Yaskawa INFORM job: A_ROOF_SIDE_0617_2_PAINT_29.JBI

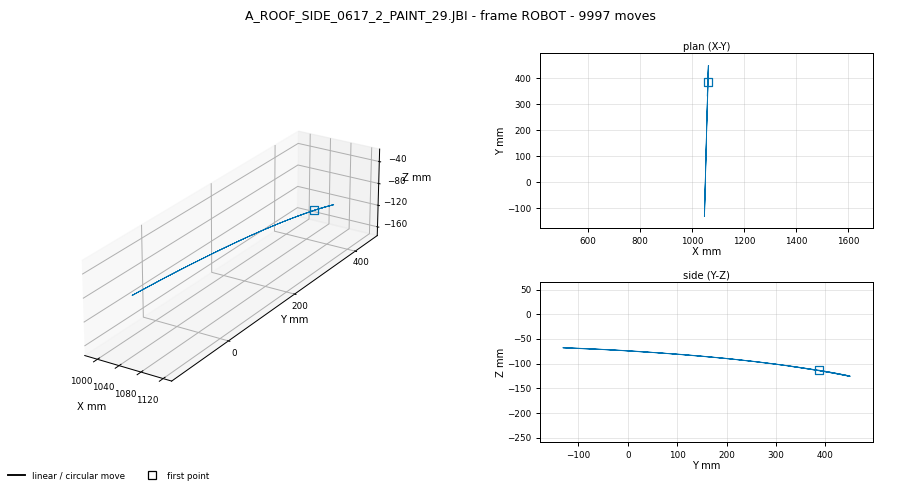
[picture p0: tool path of A_ROOF_SIDE_0617_2_PAINT_29.JBI in frame ROBOT, 9997 of 9997 moves have a stored position in this frame; points joined in program order, loops and branches not executed]
/JOB
//NAME A_ROOF_SIDE_0617_2_PAINT29
//POS
///NPOS 9997,0,0,0,0,0
///TOOL 1
///USER 0
///POSTYPE ROBOT
///RECTAN
///RCONF 1,0,0,0,0,0,0,0,0,0,0,0,0,0,0,0,0,0,0,0,0,0,0,0
C00000=1061.850,386.857,-113.195,174.714,36.908,156.968
C00001=1061.859,387.148,-113.243,174.721,36.916,156.970
C00002=1061.868,387.440,-113.291,174.727,36.924,156.972
C00003=1061.877,387.731,-113.339,174.733,36.933,156.974
C00004=1061.885,387.977,-113.380,174.739,36.940,156.976
C00005=1061.892,388.224,-113.421,174.745,36.947,156.978
C00006=1061.900,388.470,-113.462,174.750,36.954,156.979
C00007=1061.908,388.717,-113.503,174.756,36.961,156.981
C00008=1061.916,388.963,-113.543,174.761,36.968,156.983
C00009=1061.923,389.210,-113.585,174.766,36.975,156.985
C00010=1061.931,389.456,-113.625,174.773,36.983,156.986
C00011=1061.938,389.703,-113.667,174.778,36.990,156.988
C00012=1061.946,389.949,-113.707,174.783,36.997,156.990
C00013=1061.954,390.196,-113.748,174.789,37.004,156.992
C00014=1061.962,390.442,-113.789,174.794,37.012,156.994
C00015=1061.969,390.688,-113.830,174.801,37.019,156.995
C00016=1061.976,390.935,-113.872,174.806,37.026,156.997
C00017=1061.984,391.181,-113.913,174.812,37.034,156.999
C00018=1061.992,391.427,-113.954,174.817,37.041,157.001
C00019=1061.999,391.674,-113.995,174.822,37.048,157.003
C00020=1062.006,391.920,-114.037,174.829,37.056,157.005
C00021=1062.015,392.166,-114.078,174.834,37.063,157.006
C00022=1062.022,392.413,-114.119,174.840,37.071,157.008
C00023=1062.029,392.659,-114.160,174.845,37.078,157.010
C00024=1062.037,392.905,-114.202,174.852,37.086,157.012
C00025=1062.045,393.152,-114.243,174.857,37.093,157.014
C00026=1062.053,393.398,-114.285,174.863,37.100,157.016
C00027=1062.060,393.645,-114.326,174.868,37.108,157.017
C00028=1062.068,393.891,-114.368,174.875,37.116,157.019
C00029=1062.075,394.137,-114.410,174.880,37.123,157.021
C00030=1062.083,394.383,-114.452,174.886,37.131,157.023
C00031=1062.090,394.629,-114.494,174.892,37.139,157.025
C00032=1062.098,394.877,-114.535,174.898,37.146,157.027
C00033=1062.107,395.122,-114.576,174.903,37.154,157.029
C00034=1062.114,395.368,-114.618,174.910,37.161,157.031
C00035=1062.122,395.615,-114.660,174.916,37.170,157.033
C00036=1062.130,395.862,-114.702,174.921,37.177,157.035
C00037=1062.137,396.107,-114.744,174.928,37.185,157.037
C00038=1062.145,396.353,-114.786,174.933,37.192,157.039
C00039=1062.152,396.600,-114.827,174.939,37.200,157.041
C00040=1062.160,396.847,-114.869,174.945,37.208,157.042
C00041=1062.168,397.093,-114.911,174.951,37.216,157.044
C00042=1062.176,397.339,-114.954,174.957,37.223,157.046
C00043=1062.184,397.585,-114.996,174.963,37.232,157.048
C00044=1062.191,397.831,-115.038,174.969,37.240,157.050
C00045=1062.200,398.078,-115.080,174.974,37.247,157.052
C00046=1062.207,398.324,-115.122,174.981,37.255,157.054
C00047=1062.215,398.571,-115.164,174.987,37.263,157.056
C00048=1062.222,398.817,-115.207,174.993,37.271,157.058
C00049=1062.230,399.062,-115.249,174.999,37.279,157.060
C00050=1062.238,399.309,-115.292,175.005,37.287,157.062
C00051=1062.246,399.555,-115.334,175.011,37.295,157.064
C00052=1062.254,399.802,-115.376,175.017,37.303,157.066
C00053=1062.262,400.048,-115.418,175.024,37.311,157.068
C00054=1062.270,400.294,-115.461,175.029,37.319,157.070
C00055=1062.277,400.540,-115.503,175.036,37.327,157.073
C00056=1062.288,400.848,-115.556,175.043,37.337,157.075
C00057=1062.297,401.157,-115.609,175.051,37.348,157.078
C00058=1062.307,401.465,-115.663,175.059,37.358,157.080
C00059=1062.318,401.773,-115.716,175.067,37.368,157.083
C00060=1062.325,402.019,-115.760,175.073,37.376,157.085
C00061=1062.333,402.265,-115.802,175.079,37.385,157.087
C00062=1062.342,402.511,-115.845,175.086,37.393,157.089
C00063=1062.349,402.757,-115.887,175.092,37.401,157.091
C00064=1062.357,403.004,-115.930,175.099,37.410,157.094
C00065=1062.365,403.250,-115.973,175.104,37.418,157.096
C00066=1062.373,403.496,-116.015,175.111,37.426,157.098
C00067=1062.381,403.742,-116.059,175.117,37.435,157.100
C00068=1062.389,403.988,-116.102,175.124,37.443,157.102
C00069=1062.397,404.235,-116.146,175.130,37.451,157.104
C00070=1062.405,404.481,-116.188,175.136,37.460,157.106
C00071=1062.412,404.727,-116.231,175.143,37.468,157.109
C00072=1062.421,404.973,-116.274,175.149,37.477,157.111
C00073=1062.429,405.219,-116.317,175.156,37.485,157.113
C00074=1062.437,405.465,-116.361,175.162,37.494,157.115
C00075=1062.446,405.711,-116.404,175.169,37.503,157.117
C00076=1062.453,405.957,-116.447,175.176,37.511,157.120
C00077=1062.461,406.203,-116.491,175.182,37.520,157.122
C00078=1062.469,406.450,-116.534,175.188,37.529,157.124
C00079=1062.477,406.696,-116.577,175.194,37.537,157.126
C00080=1062.485,406.942,-116.620,175.201,37.546,157.129
C00081=1062.493,407.188,-116.665,175.208,37.555,157.131
C00082=1062.501,407.434,-116.708,175.215,37.564,157.133
C00083=1062.510,407.680,-116.751,175.221,37.572,157.135
C00084=1062.517,407.926,-116.795,175.228,37.581,157.138
C00085=1062.525,408.172,-116.839,175.235,37.590,157.140
C00086=1062.533,408.418,-116.882,175.241,37.599,157.142
C00087=1062.541,408.664,-116.926,175.248,37.608,157.145
C00088=1062.549,408.910,-116.970,175.255,37.616,157.147
C00089=1062.558,409.156,-117.013,175.261,37.625,157.149
C00090=1062.566,409.402,-117.058,175.268,37.634,157.151
C00091=1062.574,409.649,-117.101,175.275,37.643,157.154
C00092=1062.582,409.894,-117.146,175.282,37.652,157.156
C00093=1062.591,410.140,-117.189,175.288,37.661,157.158
C00094=1062.599,410.386,-117.233,175.295,37.670,157.161
C00095=1062.607,410.632,-117.277,175.302,37.679,157.163
C00096=1062.615,410.878,-117.320,175.310,37.688,157.165
C00097=1062.623,411.124,-117.365,175.317,37.697,157.168
C00098=1062.632,411.370,-117.409,175.323,37.706,157.170
C00099=1062.640,411.616,-117.454,175.330,37.716,157.173
C00100=1062.649,411.862,-117.497,175.337,37.725,157.175
C00101=1062.657,412.108,-117.541,175.344,37.734,157.177
C00102=1062.665,412.354,-117.586,175.351,37.743,157.180
C00103=1062.673,412.600,-117.630,175.358,37.752,157.182
C00104=1062.682,412.845,-117.674,175.365,37.762,157.185
C00105=1062.691,413.092,-117.719,175.372,37.771,157.187
C00106=1062.699,413.337,-117.763,175.379,37.780,157.190
C00107=1062.707,413.583,-117.807,175.386,37.790,157.192
C00108=1062.716,413.829,-117.851,175.394,37.799,157.194
C00109=1062.725,414.075,-117.896,175.401,37.808,157.197
C00110=1062.733,414.322,-117.941,175.408,37.818,157.199
C00111=1062.741,414.567,-117.985,175.415,37.827,157.202
C00112=1062.752,414.880,-118.042,175.424,37.839,157.205
C00113=1062.762,415.193,-118.099,175.434,37.852,157.208
C00114=1062.773,415.506,-118.156,175.443,37.864,157.212
C00115=1062.784,415.820,-118.214,175.452,37.876,157.215
C00116=1062.792,416.065,-118.258,175.460,37.886,157.217
C00117=1062.801,416.311,-118.303,175.467,37.896,157.220
C00118=1062.809,416.557,-118.348,175.474,37.905,157.223
C00119=1062.818,416.803,-118.393,175.482,37.915,157.225
C00120=1062.826,417.049,-118.438,175.489,37.925,157.228
C00121=1062.835,417.294,-118.483,175.497,37.935,157.230
C00122=1062.843,417.540,-118.528,175.504,37.945,157.233
C00123=1062.852,417.786,-118.573,175.511,37.954,157.236
C00124=1062.860,418.031,-118.618,175.519,37.964,157.238
C00125=1062.869,418.277,-118.664,175.526,37.974,157.241
C00126=1062.878,418.524,-118.709,175.534,37.984,157.243
C00127=1062.886,418.769,-118.754,175.541,37.994,157.246
C00128=1062.895,419.015,-118.799,175.549,38.004,157.249
C00129=1062.903,419.261,-118.845,175.557,38.014,157.251
C00130=1062.912,419.506,-118.890,175.565,38.024,157.254
C00131=1062.920,419.752,-118.935,175.572,38.034,157.257
C00132=1062.929,419.998,-118.981,175.580,38.043,157.259
C00133=1062.938,420.243,-119.026,175.587,38.054,157.262
C00134=1062.947,420.489,-119.072,175.595,38.064,157.265
C00135=1062.955,420.735,-119.117,175.604,38.074,157.268
C00136=1062.964,420.980,-119.163,175.611,38.084,157.270
C00137=1062.973,421.226,-119.210,175.619,38.095,157.273
C00138=1062.982,421.472,-119.255,175.626,38.105,157.276
C00139=1062.991,421.718,-119.300,175.635,38.116,157.279
C00140=1062.998,421.962,-119.347,175.643,38.125,157.282
C00141=1063.007,422.208,-119.392,175.650,38.136,157.284
C00142=1063.016,422.454,-119.438,175.658,38.146,157.287
C00143=1063.025,422.700,-119.484,175.666,38.157,157.290
C00144=1063.033,422.946,-119.530,175.674,38.167,157.293
C00145=1063.043,423.191,-119.576,175.682,38.178,157.296
C00146=1063.051,423.436,-119.623,175.691,38.188,157.299
C00147=1063.060,423.682,-119.669,175.698,38.199,157.301
C00148=1063.069,423.927,-119.715,175.706,38.210,157.304
C00149=1063.078,424.173,-119.761,175.715,38.220,157.307
C00150=1063.087,424.419,-119.807,175.723,38.230,157.310
C00151=1063.095,424.664,-119.854,175.731,38.241,157.313
C00152=1063.105,424.910,-119.900,175.739,38.252,157.316
C00153=1063.113,425.155,-119.946,175.747,38.263,157.319
C00154=1063.122,425.400,-119.993,175.756,38.274,157.322
C00155=1063.131,425.646,-120.039,175.764,38.284,157.325
C00156=1063.140,425.891,-120.085,175.773,38.295,157.328
C00157=1063.149,426.137,-120.133,175.780,38.306,157.331
C00158=1063.159,426.382,-120.179,175.789,38.317,157.334
C00159=1063.167,426.628,-120.225,175.797,38.328,157.337
C00160=1063.177,426.873,-120.272,175.806,38.339,157.340
C00161=1063.185,427.119,-120.318,175.814,38.350,157.343
C00162=1063.194,427.365,-120.365,175.823,38.361,157.346
C00163=1063.203,427.610,-120.413,175.831,38.372,157.349
C00164=1063.212,427.855,-120.459,175.840,38.383,157.352
C00165=1063.221,428.100,-120.506,175.849,38.394,157.355
C00166=1063.230,428.346,-120.554,175.857,38.405,157.358
C00167=1063.239,428.592,-120.600,175.866,38.417,157.361
C00168=1063.252,428.924,-120.664,175.877,38.432,157.365
C00169=1063.264,429.258,-120.728,175.889,38.447,157.370
C00170=1063.276,429.591,-120.792,175.902,38.463,157.374
C00171=1063.289,429.925,-120.856,175.913,38.478,157.378
C00172=1063.298,430.170,-120.904,175.922,38.489,157.381
C00173=1063.308,430.415,-120.951,175.931,38.501,157.384
C00174=1063.316,430.661,-120.998,175.940,38.512,157.388
C00175=1063.326,430.906,-121.046,175.948,38.524,157.391
C00176=1063.334,431.151,-121.093,175.958,38.536,157.394
C00177=1063.344,431.397,-121.141,175.967,38.547,157.397
C00178=1063.353,431.642,-121.189,175.976,38.559,157.401
C00179=1063.362,431.887,-121.237,175.984,38.570,157.404
C00180=1063.371,432.132,-121.284,175.993,38.582,157.407
C00181=1063.381,432.377,-121.332,176.003,38.594,157.411
C00182=1063.390,432.623,-121.380,176.012,38.606,157.414
C00183=1063.399,432.868,-121.428,176.021,38.618,157.417
C00184=1063.409,433.113,-121.476,176.031,38.629,157.420
C00185=1063.418,433.358,-121.524,176.040,38.641,157.424
C00186=1063.427,433.603,-121.572,176.049,38.653,157.427
C00187=1063.437,433.849,-121.619,176.059,38.665,157.431
C00188=1063.446,434.094,-121.668,176.068,38.677,157.434
C00189=1063.455,434.339,-121.715,176.077,38.689,157.437
C00190=1063.465,434.584,-121.764,176.087,38.701,157.441
C00191=1063.475,434.829,-121.812,176.096,38.714,157.444
C00192=1063.484,435.074,-121.860,176.106,38.726,157.448
C00193=1063.493,435.318,-121.908,176.115,38.738,157.451
C00194=1063.502,435.564,-121.957,176.124,38.750,157.454
C00195=1063.512,435.809,-122.005,176.134,38.763,157.458
C00196=1063.522,436.054,-122.054,176.144,38.775,157.462
C00197=1063.531,436.299,-122.102,176.153,38.787,157.465
C00198=1063.541,436.544,-122.151,176.163,38.799,157.469
C00199=1063.551,436.789,-122.199,176.173,38.812,157.472
C00200=1063.561,437.034,-122.248,176.183,38.824,157.476
C00201=1063.570,437.279,-122.296,176.192,38.837,157.479
C00202=1063.579,437.524,-122.346,176.202,38.849,157.483
C00203=1063.589,437.769,-122.394,176.212,38.862,157.486
C00204=1063.599,438.014,-122.443,176.222,38.874,157.490
C00205=1063.609,438.259,-122.492,176.232,38.887,157.494
C00206=1063.618,438.504,-122.541,176.242,38.900,157.497
C00207=1063.628,438.749,-122.589,176.251,38.912,157.501
C00208=1063.639,438.994,-122.639,176.262,38.925,157.505
C00209=1063.648,439.239,-122.688,176.272,38.938,157.508
C00210=1063.658,439.484,-122.737,176.282,38.951,157.512
C00211=1063.667,439.729,-122.786,176.292,38.964,157.516
C00212=1063.677,439.973,-122.836,176.302,38.977,157.520
C00213=1063.687,440.218,-122.885,176.313,38.990,157.523
C00214=1063.696,440.464,-122.935,176.323,39.003,157.527
C00215=1063.706,440.708,-122.984,176.334,39.016,157.531
C00216=1063.717,440.952,-123.033,176.344,39.029,157.535
C00217=1063.726,441.198,-123.083,176.354,39.042,157.538
C00218=1063.737,441.442,-123.132,176.364,39.056,157.542
C00219=1063.746,441.687,-123.182,176.375,39.069,157.546
C00220=1063.756,441.932,-123.232,176.385,39.082,157.550
C00221=1063.766,442.176,-123.282,176.396,39.095,157.554
C00222=1063.776,442.421,-123.331,176.407,39.109,157.558
C00223=1063.786,442.666,-123.381,176.417,39.122,157.562
C00224=1063.800,442.997,-123.449,176.432,39.141,157.567
C00225=1063.813,443.330,-123.517,176.446,39.159,157.573
C00226=1063.827,443.662,-123.585,176.461,39.177,157.578
C00227=1063.841,443.993,-123.652,176.477,39.196,157.583
C00228=1063.851,444.238,-123.703,176.487,39.209,157.587
C00229=1063.860,444.483,-123.753,176.498,39.223,157.592
C00230=1063.871,444.727,-123.804,176.509,39.237,157.596
C00231=1063.881,444.972,-123.854,176.520,39.251,157.600
C00232=1063.891,445.217,-123.904,176.532,39.265,157.604
C00233=1063.902,445.461,-123.955,176.543,39.279,157.608
C00234=1063.912,445.706,-124.006,176.554,39.293,157.612
C00235=1063.922,445.950,-124.056,176.566,39.307,157.616
C00236=1063.932,446.194,-124.106,176.576,39.321,157.620
C00237=1063.943,446.439,-124.157,176.588,39.335,157.625
C00238=1063.953,446.684,-124.208,176.600,39.349,157.629
C00239=1063.963,446.929,-124.259,176.611,39.364,157.633
C00240=1063.974,447.172,-124.310,176.622,39.378,157.637
C00241=1063.984,447.415,-124.360,176.634,39.392,157.642
C00242=1063.995,447.660,-124.411,176.645,39.406,157.646
C00243=1064.006,447.904,-124.461,176.657,39.420,157.650
C00244=1064.019,448.147,-124.510,176.669,39.434,157.654
C00245=1064.032,448.391,-124.559,176.681,39.447,157.658
C00246=1064.046,448.636,-124.607,176.693,39.460,157.662
C00247=1064.062,448.881,-124.655,176.704,39.473,157.666
C00248=1064.078,449.126,-124.702,176.716,39.486,157.670
C00249=1064.096,449.371,-124.748,176.729,39.498,157.674
C00250=1064.114,449.616,-124.793,176.740,39.510,157.677
C00251=1064.133,449.862,-124.838,176.752,39.522,157.681
C00252=1063.796,449.868,-125.107,176.744,39.644,157.714
C00253=1063.776,449.622,-125.063,176.733,39.632,157.711
C00254=1063.758,449.378,-125.017,176.720,39.621,157.707
C00255=1063.740,449.132,-124.971,176.708,39.608,157.703
C00256=1063.724,448.888,-124.924,176.696,39.596,157.699
C00257=1063.709,448.643,-124.877,176.684,39.583,157.695
C00258=1063.693,448.398,-124.828,176.672,39.570,157.691
C00259=1063.680,448.154,-124.780,176.660,39.557,157.687
C00260=1063.668,447.911,-124.731,176.648,39.543,157.683
C00261=1063.657,447.694,-124.686,176.637,39.531,157.679
C00262=1063.648,447.478,-124.642,176.627,39.518,157.676
C00263=1063.638,447.262,-124.596,176.617,39.506,157.672
C00264=1063.629,447.047,-124.551,176.606,39.493,157.668
C00265=1063.620,446.830,-124.507,176.596,39.480,157.664
C00266=1063.611,446.615,-124.462,176.586,39.468,157.661
C00267=1063.601,446.399,-124.417,176.576,39.455,157.657
C00268=1063.592,446.184,-124.372,176.566,39.443,157.653
C00269=1063.582,445.939,-124.321,176.555,39.429,157.649
C00270=1063.571,445.695,-124.271,176.543,39.415,157.645
C00271=1063.561,445.450,-124.220,176.532,39.401,157.641
C00272=1063.552,445.205,-124.170,176.521,39.387,157.637
C00273=1063.541,444.961,-124.120,176.510,39.373,157.632
C00274=1063.530,444.716,-124.069,176.498,39.360,157.628
C00275=1063.521,444.472,-124.018,176.487,39.346,157.624
C00276=1063.510,444.227,-123.969,176.476,39.332,157.620
C00277=1063.495,443.858,-123.892,176.459,39.311,157.614
C00278=1063.480,443.489,-123.817,176.442,39.291,157.608
C00279=1063.464,443.120,-123.741,176.427,39.271,157.602
C00280=1063.449,442.750,-123.665,176.410,39.250,157.596
C00281=1063.439,442.505,-123.616,176.399,39.237,157.592
C00282=1063.429,442.260,-123.566,176.389,39.224,157.588
C00283=1063.419,442.016,-123.516,176.378,39.210,157.584
C00284=1063.409,441.771,-123.465,176.367,39.197,157.580
C00285=1063.399,441.527,-123.416,176.357,39.184,157.576
C00286=1063.390,441.282,-123.366,176.346,39.170,157.573
C00287=1063.379,441.037,-123.317,176.335,39.157,157.569
C00288=1063.370,440.792,-123.267,176.325,39.144,157.565
C00289=1063.360,440.547,-123.218,176.314,39.131,157.561
C00290=1063.349,440.302,-123.169,176.304,39.118,157.557
C00291=1063.340,440.058,-123.119,176.294,39.105,157.554
C00292=1063.330,439.813,-123.070,176.284,39.092,157.550
C00293=1063.320,439.567,-123.020,176.273,39.080,157.546
C00294=1063.310,439.323,-122.971,176.263,39.066,157.542
C00295=1063.300,439.078,-122.922,176.252,39.054,157.539
C00296=1063.291,438.833,-122.873,176.243,39.041,157.535
C00297=1063.281,438.588,-122.824,176.233,39.028,157.531
C00298=1063.271,438.344,-122.775,176.222,39.015,157.527
C00299=1063.262,438.099,-122.726,176.212,39.003,157.524
C00300=1063.252,437.854,-122.676,176.203,38.990,157.520
C00301=1063.242,437.609,-122.628,176.192,38.978,157.517
C00302=1063.232,437.364,-122.579,176.182,38.965,157.513
C00303=1063.222,437.119,-122.530,176.173,38.952,157.509
C00304=1063.212,436.874,-122.482,176.162,38.940,157.506
C00305=1063.203,436.628,-122.433,176.153,38.928,157.502
C00306=1063.194,436.383,-122.384,176.143,38.915,157.499
C00307=1063.184,436.138,-122.336,176.134,38.903,157.495
C00308=1063.174,435.894,-122.287,176.124,38.891,157.492
C00309=1063.164,435.649,-122.239,176.114,38.879,157.488
C00310=1063.155,435.404,-122.190,176.104,38.867,157.485
C00311=1063.145,435.158,-122.142,176.094,38.854,157.481
C00312=1063.136,434.914,-122.094,176.085,38.842,157.478
C00313=1063.126,434.669,-122.046,176.076,38.830,157.474
C00314=1063.117,434.423,-121.998,176.066,38.818,157.471
C00315=1063.107,434.178,-121.949,176.057,38.806,157.468
C00316=1063.098,433.933,-121.900,176.047,38.794,157.464
C00317=1063.089,433.688,-121.853,176.038,38.782,157.461
C00318=1063.079,433.443,-121.804,176.029,38.770,157.457
C00319=1063.070,433.197,-121.756,176.019,38.759,157.454
C00320=1063.061,432.953,-121.709,176.010,38.746,157.451
C00321=1063.051,432.708,-121.661,176.001,38.735,157.447
C00322=1063.042,432.462,-121.613,175.991,38.723,157.444
C00323=1063.033,432.217,-121.565,175.982,38.711,157.441
C00324=1063.024,431.971,-121.517,175.973,38.699,157.437
C00325=1063.014,431.727,-121.469,175.964,38.688,157.434
C00326=1063.005,431.482,-121.421,175.954,38.676,157.431
C00327=1062.996,431.236,-121.374,175.945,38.664,157.428
C00328=1062.987,430.991,-121.326,175.937,38.653,157.424
C00329=1062.977,430.746,-121.278,175.928,38.641,157.421
C00330=1062.968,430.501,-121.231,175.919,38.630,157.418
C00331=1062.959,430.255,-121.184,175.909,38.619,157.415
C00332=1062.950,430.010,-121.137,175.900,38.607,157.411
C00333=1062.937,429.675,-121.072,175.889,38.592,157.407
C00334=1062.924,429.339,-121.008,175.877,38.576,157.403
C00335=1062.912,429.004,-120.943,175.864,38.561,157.399
C00336=1062.899,428.668,-120.878,175.852,38.545,157.394
C00337=1062.890,428.423,-120.832,175.844,38.534,157.391
C00338=1062.882,428.178,-120.784,175.835,38.523,157.388
C00339=1062.872,427.932,-120.738,175.826,38.512,157.385
C00340=1062.863,427.687,-120.690,175.818,38.501,157.382
C00341=1062.854,427.442,-120.643,175.809,38.490,157.379
C00342=1062.846,427.196,-120.597,175.801,38.479,157.376
C00343=1062.836,426.951,-120.549,175.792,38.468,157.373
C00344=1062.827,426.705,-120.503,175.784,38.457,157.370
C00345=1062.818,426.460,-120.457,175.775,38.446,157.367
C00346=1062.809,426.215,-120.410,175.766,38.435,157.364
C00347=1062.801,425.969,-120.363,175.759,38.424,157.361
C00348=1062.791,425.723,-120.317,175.750,38.414,157.358
C00349=1062.782,425.478,-120.270,175.742,38.403,157.355
C00350=1062.773,425.233,-120.224,175.733,38.392,157.352
C00351=1062.764,424.987,-120.178,175.725,38.382,157.349
C00352=1062.755,424.742,-120.131,175.716,38.371,157.346
C00353=1062.746,424.497,-120.085,175.708,38.360,157.343
C00354=1062.737,424.251,-120.038,175.700,38.349,157.340
C00355=1062.728,424.005,-119.993,175.692,38.339,157.337
C00356=1062.720,423.760,-119.946,175.684,38.328,157.334
C00357=1062.710,423.515,-119.900,175.675,38.318,157.332
C00358=1062.702,423.268,-119.854,175.668,38.307,157.329
C00359=1062.693,423.023,-119.808,175.660,38.297,157.326
C00360=1062.684,422.778,-119.761,175.651,38.286,157.323
C00361=1062.675,422.532,-119.715,175.644,38.276,157.320
C00362=1062.666,422.287,-119.669,175.635,38.265,157.317
C00363=1062.658,422.041,-119.623,175.627,38.255,157.315
C00364=1062.649,421.795,-119.577,175.620,38.245,157.312
C00365=1062.640,421.549,-119.531,175.611,38.235,157.309
C00366=1062.631,421.303,-119.486,175.603,38.224,157.306
C00367=1062.623,421.059,-119.439,175.596,38.214,157.303
C00368=1062.614,420.813,-119.394,175.588,38.204,157.301
C00369=1062.605,420.567,-119.349,175.580,38.193,157.298
C00370=1062.597,420.321,-119.303,175.572,38.183,157.295
C00371=1062.588,420.075,-119.257,175.564,38.174,157.292
C00372=1062.579,419.829,-119.212,175.557,38.163,157.290
C00373=1062.571,419.584,-119.167,175.548,38.153,157.287
C00374=1062.562,419.338,-119.121,175.541,38.143,157.284
C00375=1062.554,419.092,-119.075,175.533,38.133,157.282
C00376=1062.545,418.846,-119.030,175.526,38.123,157.279
C00377=1062.536,418.601,-118.985,175.518,38.113,157.276
C00378=1062.527,418.355,-118.939,175.511,38.103,157.273
C00379=1062.518,418.110,-118.894,175.502,38.094,157.271
C00380=1062.510,417.864,-118.849,175.495,38.084,157.268
C00381=1062.501,417.618,-118.804,175.487,38.074,157.266
C00382=1062.493,417.373,-118.759,175.480,38.064,157.263
C00383=1062.485,417.127,-118.713,175.473,38.055,157.260
C00384=1062.476,416.880,-118.668,175.465,38.045,157.258
C00385=1062.468,416.635,-118.623,175.458,38.035,157.255
C00386=1062.459,416.389,-118.578,175.450,38.025,157.253
C00387=1062.451,416.144,-118.534,175.443,38.016,157.250
C00388=1062.442,415.898,-118.488,175.436,38.006,157.247
C00389=1062.432,415.583,-118.431,175.426,37.994,157.244
C00390=1062.420,415.268,-118.374,175.416,37.981,157.241
C00391=1062.410,414.953,-118.316,175.407,37.969,157.238
C00392=1062.399,414.638,-118.259,175.398,37.957,157.234
C00393=1062.391,414.392,-118.214,175.390,37.948,157.232
C00394=1062.383,414.146,-118.169,175.383,37.938,157.229
C00395=1062.373,413.900,-118.125,175.376,37.929,157.227
C00396=1062.365,413.654,-118.081,175.369,37.920,157.225
C00397=1062.356,413.408,-118.036,175.362,37.910,157.222
C00398=1062.348,413.162,-117.992,175.355,37.901,157.220
C00399=1062.340,412.916,-117.948,175.348,37.892,157.217
C00400=1062.331,412.670,-117.904,175.341,37.882,157.215
C00401=1062.323,412.424,-117.859,175.333,37.873,157.212
C00402=1062.315,412.179,-117.815,175.326,37.864,157.210
C00403=1062.306,411.932,-117.770,175.319,37.855,157.207
C00404=1062.297,411.687,-117.726,175.312,37.846,157.205
C00405=1062.289,411.441,-117.682,175.305,37.836,157.203
C00406=1062.281,411.195,-117.638,175.298,37.827,157.200
C00407=1062.273,410.949,-117.594,175.292,37.818,157.198
C00408=1062.264,410.703,-117.550,175.284,37.809,157.195
C00409=1062.256,410.457,-117.506,175.277,37.800,157.193
C00410=1062.248,410.211,-117.462,175.270,37.791,157.191
C00411=1062.239,409.965,-117.418,175.263,37.782,157.188
C00412=1062.231,409.719,-117.374,175.257,37.773,157.186
C00413=1062.223,409.473,-117.330,175.250,37.764,157.184
C00414=1062.215,409.227,-117.286,175.243,37.755,157.181
C00415=1062.206,408.981,-117.243,175.236,37.746,157.179
C00416=1062.198,408.735,-117.198,175.229,37.738,157.177
C00417=1062.190,408.488,-117.155,175.223,37.729,157.174
C00418=1062.182,408.243,-117.111,175.216,37.720,157.172
C00419=1062.174,407.997,-117.067,175.209,37.711,157.170
C00420=1062.166,407.750,-117.024,175.202,37.702,157.168
C00421=1062.157,407.505,-116.980,175.196,37.694,157.165
C00422=1062.150,407.259,-116.936,175.189,37.685,157.163
C00423=1062.142,407.013,-116.893,175.182,37.676,157.161
C00424=1062.134,406.767,-116.850,175.176,37.668,157.159
C00425=1062.126,406.520,-116.806,175.169,37.659,157.156
C00426=1062.117,406.275,-116.763,175.162,37.650,157.154
C00427=1062.110,406.029,-116.719,175.156,37.642,157.152
C00428=1062.102,405.782,-116.675,175.150,37.633,157.150
C00429=1062.093,405.536,-116.632,175.143,37.624,157.147
C00430=1062.086,405.290,-116.589,175.137,37.616,157.145
C00431=1062.078,405.045,-116.546,175.130,37.607,157.143
C00432=1062.069,404.798,-116.503,175.123,37.599,157.141
C00433=1062.061,404.552,-116.459,175.117,37.591,157.139
C00434=1062.053,404.306,-116.416,175.110,37.582,157.136
C00435=1062.045,404.059,-116.374,175.104,37.574,157.134
C00436=1062.038,403.814,-116.331,175.098,37.565,157.132
C00437=1062.030,403.567,-116.287,175.091,37.557,157.130
C00438=1062.021,403.321,-116.244,175.085,37.548,157.128
C00439=1062.013,403.075,-116.202,175.078,37.540,157.126
C00440=1062.006,402.829,-116.159,175.072,37.532,157.123
C00441=1061.997,402.583,-116.116,175.066,37.523,157.121
C00442=1061.989,402.336,-116.073,175.059,37.515,157.119
C00443=1061.982,402.091,-116.030,175.053,37.507,157.117
C00444=1061.974,401.844,-115.988,175.046,37.499,157.115
C00445=1061.964,401.534,-115.934,175.038,37.489,157.112
C00446=1061.954,401.224,-115.880,175.031,37.478,157.110
C00447=1061.944,400.914,-115.827,175.023,37.468,157.107
C00448=1061.933,400.604,-115.773,175.016,37.458,157.105
C00449=1061.925,400.358,-115.730,175.009,37.450,157.102
C00450=1061.918,400.112,-115.688,175.003,37.441,157.100
C00451=1061.910,399.865,-115.646,174.996,37.433,157.098
C00452=1061.902,399.620,-115.603,174.991,37.425,157.096
C00453=1061.894,399.373,-115.561,174.984,37.418,157.094
C00454=1061.886,399.127,-115.519,174.978,37.410,157.092
C00455=1061.878,398.881,-115.476,174.972,37.402,157.090
C00456=1061.870,398.635,-115.434,174.966,37.394,157.088
C00457=1061.863,398.388,-115.391,174.959,37.386,157.086
C00458=1061.855,398.142,-115.349,174.954,37.378,157.084
C00459=1061.847,397.896,-115.306,174.948,37.370,157.082
C00460=1061.839,397.650,-115.265,174.942,37.362,157.080
C00461=1061.832,397.404,-115.223,174.936,37.354,157.078
C00462=1061.823,397.157,-115.180,174.929,37.346,157.076
C00463=1061.816,396.911,-115.138,174.924,37.339,157.074
C00464=1061.808,396.664,-115.096,174.918,37.331,157.072
C00465=1061.800,396.418,-115.055,174.912,37.323,157.070
C00466=1061.793,396.172,-115.013,174.906,37.315,157.068
C00467=1061.785,395.925,-114.971,174.899,37.308,157.066
C00468=1061.777,395.679,-114.929,174.894,37.300,157.065
C00469=1061.769,395.433,-114.887,174.888,37.293,157.063
C00470=1061.762,395.187,-114.845,174.882,37.284,157.061
C00471=1061.753,394.940,-114.804,174.876,37.277,157.059
C00472=1061.746,394.694,-114.762,174.871,37.269,157.057
C00473=1061.738,394.448,-114.721,174.864,37.262,157.055
C00474=1061.731,394.202,-114.679,174.859,37.254,157.053
C00475=1061.723,393.955,-114.636,174.853,37.247,157.051
C00476=1061.715,393.708,-114.595,174.847,37.239,157.049
C00477=1061.708,393.462,-114.553,174.841,37.232,157.047
C00478=1061.700,393.216,-114.512,174.836,37.224,157.046
C00479=1061.692,392.970,-114.471,174.829,37.216,157.044
C00480=1061.685,392.724,-114.429,174.824,37.209,157.042
C00481=1061.677,392.477,-114.387,174.818,37.202,157.040
C00482=1061.669,392.230,-114.346,174.813,37.194,157.038
C00483=1061.661,391.984,-114.305,174.806,37.187,157.036
C00484=1061.654,391.738,-114.263,174.801,37.179,157.034
C00485=1061.646,391.492,-114.222,174.795,37.172,157.033
C00486=1061.639,391.245,-114.181,174.789,37.164,157.031
C00487=1061.631,390.999,-114.139,174.783,37.157,157.029
C00488=1061.623,390.753,-114.098,174.778,37.150,157.027
C00489=1061.616,390.506,-114.057,174.773,37.143,157.025
C00490=1061.608,390.260,-114.016,174.766,37.135,157.023
C00491=1061.601,390.013,-113.975,174.761,37.128,157.022
C00492=1061.593,389.767,-113.934,174.755,37.121,157.020
C00493=1061.586,389.520,-113.893,174.750,37.114,157.018
C00494=1061.578,389.274,-113.853,174.745,37.106,157.016
C00495=1061.570,389.027,-113.811,174.738,37.099,157.014
C00496=1061.562,388.781,-113.771,174.733,37.092,157.013
C00497=1061.555,388.535,-113.729,174.727,37.085,157.011
C00498=1061.547,388.288,-113.689,174.722,37.078,157.009
C00499=1061.540,388.042,-113.648,174.717,37.071,157.007
C00500=1061.532,387.795,-113.607,174.710,37.064,157.006
C00501=1061.523,387.502,-113.558,174.704,37.055,157.004
C00502=1061.514,387.210,-113.511,174.698,37.047,157.001
C00503=1061.505,386.917,-113.461,174.691,37.039,156.999
C00504=1061.496,386.623,-113.413,174.685,37.030,156.997
C00505=1061.488,386.377,-113.373,174.679,37.023,156.996
C00506=1061.480,386.130,-113.331,174.674,37.016,156.994
C00507=1061.473,385.884,-113.292,174.668,37.009,156.992
C00508=1061.465,385.638,-113.251,174.663,37.002,156.990
C00509=1061.458,385.390,-113.211,174.657,36.996,156.989
C00510=1061.450,385.144,-113.170,174.652,36.988,156.987
C00511=1061.444,384.898,-113.129,174.647,36.981,156.985
C00512=1061.436,384.651,-113.089,174.641,36.975,156.984
C00513=1061.428,384.405,-113.049,174.636,36.968,156.982
C00514=1061.421,384.158,-113.008,174.631,36.961,156.980
C00515=1061.413,383.912,-112.968,174.626,36.954,156.979
C00516=1061.406,383.665,-112.927,174.619,36.947,156.977
C00517=1061.399,383.418,-112.887,174.614,36.940,156.975
C00518=1061.391,383.173,-112.847,174.609,36.933,156.974
C00519=1061.384,382.925,-112.807,174.604,36.927,156.972
C00520=1061.377,382.678,-112.767,174.599,36.920,156.970
C00521=1061.369,382.433,-112.726,174.593,36.913,156.969
C00522=1061.362,382.186,-112.686,174.588,36.906,156.967
C00523=1061.355,381.939,-112.646,174.583,36.899,156.965
C00524=1061.347,381.693,-112.606,174.578,36.893,156.964
C00525=1061.340,381.446,-112.565,174.573,36.886,156.962
C00526=1061.333,381.200,-112.526,174.568,36.879,156.960
C00527=1061.325,380.953,-112.486,174.562,36.873,156.959
C00528=1061.318,380.706,-112.445,174.557,36.866,156.957
C00529=1061.311,380.459,-112.406,174.552,36.859,156.956
C00530=1061.303,380.212,-112.366,174.546,36.853,156.954
C00531=1061.296,379.966,-112.326,174.541,36.846,156.952
C00532=1061.289,379.719,-112.286,174.536,36.840,156.951
C00533=1061.281,379.472,-112.246,174.530,36.833,156.949
C00534=1061.274,379.226,-112.207,174.525,36.826,156.948
C00535=1061.266,378.979,-112.167,174.520,36.820,156.946
C00536=1061.259,378.733,-112.127,174.515,36.813,156.945
C00537=1061.251,378.486,-112.087,174.510,36.807,156.943
C00538=1061.244,378.239,-112.048,174.505,36.801,156.941
C00539=1061.237,377.993,-112.009,174.500,36.794,156.940
C00540=1061.230,377.746,-111.969,174.495,36.787,156.938
C00541=1061.222,377.499,-111.929,174.490,36.781,156.937
C00542=1061.215,377.253,-111.890,174.484,36.775,156.935
C00543=1061.207,377.006,-111.850,174.479,36.768,156.934
C00544=1061.200,376.759,-111.811,174.475,36.762,156.932
C00545=1061.193,376.513,-111.771,174.470,36.756,156.931
C00546=1061.186,376.266,-111.732,174.465,36.749,156.929
C00547=1061.179,376.020,-111.692,174.460,36.743,156.928
C00548=1061.171,375.772,-111.653,174.455,36.736,156.926
C00549=1061.164,375.526,-111.614,174.450,36.730,156.925
C00550=1061.157,375.279,-111.575,174.445,36.724,156.923
C00551=1061.149,375.032,-111.535,174.440,36.718,156.921
C00552=1061.143,374.785,-111.496,174.435,36.711,156.920
C00553=1061.136,374.539,-111.457,174.430,36.705,156.918
C00554=1061.128,374.292,-111.417,174.425,36.698,156.917
C00555=1061.121,374.045,-111.378,174.420,36.692,156.915
C00556=1061.114,373.799,-111.339,174.415,36.686,156.914
C00557=1061.107,373.537,-111.297,174.410,36.680,156.912
C00558=1061.099,373.274,-111.256,174.404,36.673,156.911
C00559=1061.092,373.012,-111.214,174.399,36.666,156.909
C00560=1061.084,372.751,-111.173,174.394,36.660,156.908
C00561=1061.076,372.503,-111.134,174.389,36.653,156.906
C00562=1061.069,372.257,-111.095,174.384,36.647,156.905
C00563=1061.062,372.010,-111.056,174.379,36.641,156.903
C00564=1061.056,371.763,-111.017,174.375,36.635,156.902
C00565=1061.048,371.516,-110.978,174.370,36.629,156.900
C00566=1061.041,371.269,-110.940,174.365,36.623,156.899
C00567=1061.033,371.023,-110.901,174.360,36.617,156.897
C00568=1061.026,370.776,-110.862,174.355,36.610,156.896
C00569=1061.019,370.529,-110.823,174.350,36.604,156.894
C00570=1061.011,370.282,-110.784,174.345,36.598,156.893
C00571=1061.004,370.035,-110.745,174.341,36.593,156.892
C00572=1060.997,369.788,-110.707,174.337,36.587,156.890
C00573=1060.990,369.541,-110.669,174.332,36.580,156.889
C00574=1060.983,369.294,-110.630,174.327,36.574,156.887
C00575=1060.976,369.047,-110.591,174.322,36.568,156.886
C00576=1060.968,368.800,-110.553,174.317,36.562,156.884
C00577=1060.962,368.554,-110.514,174.312,36.557,156.883
C00578=1060.954,368.307,-110.476,174.307,36.551,156.882
C00579=1060.947,368.060,-110.437,174.303,36.544,156.880
C00580=1060.941,367.813,-110.399,174.298,36.539,156.879
C00581=1060.933,367.566,-110.361,174.294,36.533,156.878
C00582=1060.926,367.319,-110.322,174.289,36.527,156.876
C00583=1060.919,367.073,-110.283,174.284,36.521,156.875
C00584=1060.912,366.826,-110.245,174.279,36.515,156.873
C00585=1060.906,366.579,-110.207,174.275,36.509,156.872
C00586=1060.898,366.332,-110.168,174.270,36.503,156.871
C00587=1060.891,366.085,-110.130,174.265,36.497,156.869
C00588=1060.884,365.838,-110.092,174.261,36.492,156.868
C00589=1060.877,365.591,-110.054,174.256,36.486,156.866
C00590=1060.870,365.344,-110.016,174.252,36.480,156.865
C00591=1060.863,365.097,-109.977,174.247,36.474,156.864
C00592=1060.856,364.850,-109.939,174.242,36.468,156.862
C00593=1060.849,364.603,-109.901,174.238,36.462,156.861
C00594=1060.842,364.356,-109.862,174.233,36.457,156.860
C00595=1060.835,364.109,-109.825,174.229,36.451,156.858
C00596=1060.828,363.862,-109.786,174.224,36.445,156.857
C00597=1060.821,363.615,-109.748,174.219,36.439,156.856
C00598=1060.814,363.368,-109.711,174.215,36.434,156.854
C00599=1060.807,363.121,-109.672,174.210,36.428,156.853
C00600=1060.800,362.875,-109.635,174.206,36.422,156.852
C00601=1060.793,362.627,-109.597,174.201,36.416,156.850
C00602=1060.786,362.380,-109.560,174.197,36.411,156.849
C00603=1060.779,362.133,-109.521,174.192,36.405,156.848
C00604=1060.772,361.886,-109.483,174.188,36.400,156.846
C00605=1060.765,361.639,-109.446,174.183,36.394,156.845
C00606=1060.758,361.392,-109.408,174.178,36.389,156.844
C00607=1060.751,361.145,-109.370,174.174,36.383,156.842
C00608=1060.744,360.898,-109.333,174.170,36.377,156.841
C00609=1060.737,360.652,-109.295,174.165,36.372,156.840
C00610=1060.730,360.407,-109.258,174.161,36.366,156.839
C00611=1060.723,360.162,-109.220,174.156,36.361,156.837
C00612=1060.716,359.916,-109.183,174.152,36.355,156.836
C00613=1060.709,359.671,-109.146,174.147,36.349,156.835
C00614=1060.703,359.425,-109.108,174.143,36.344,156.833
C00615=1060.696,359.180,-109.072,174.138,36.339,156.832
C00616=1060.689,358.934,-109.034,174.134,36.333,156.831
C00617=1060.681,358.687,-108.996,174.130,36.328,156.830
C00618=1060.675,358.441,-108.959,174.125,36.322,156.828
C00619=1060.668,358.193,-108.921,174.120,36.316,156.827
C00620=1060.661,357.945,-108.884,174.117,36.311,156.826
C00621=1060.655,357.699,-108.847,174.112,36.306,156.825
C00622=1060.647,357.452,-108.809,174.107,36.300,156.823
C00623=1060.640,357.205,-108.772,174.104,36.294,156.822
C00624=1060.633,356.958,-108.734,174.099,36.289,156.821
C00625=1060.627,356.711,-108.698,174.094,36.284,156.819
C00626=1060.619,356.463,-108.660,174.091,36.279,156.818
C00627=1060.612,356.216,-108.623,174.086,36.273,156.817
C00628=1060.606,355.969,-108.586,174.081,36.268,156.816
C00629=1060.598,355.722,-108.549,174.077,36.262,156.815
C00630=1060.592,355.474,-108.512,174.073,36.257,156.813
C00631=1060.585,355.228,-108.475,174.068,36.252,156.812
C00632=1060.578,354.981,-108.437,174.064,36.246,156.811
C00633=1060.571,354.733,-108.401,174.060,36.241,156.810
C00634=1060.564,354.487,-108.363,174.056,36.235,156.808
C00635=1060.557,354.239,-108.327,174.051,36.230,156.807
C00636=1060.550,353.992,-108.289,174.047,36.225,156.806
C00637=1060.544,353.745,-108.253,174.043,36.220,156.805
C00638=1060.537,353.498,-108.215,174.038,36.214,156.803
C00639=1060.530,353.250,-108.179,174.035,36.209,156.802
C00640=1060.523,353.003,-108.142,174.030,36.203,156.801
C00641=1060.516,352.756,-108.105,174.025,36.198,156.800
C00642=1060.509,352.509,-108.068,174.022,36.193,156.799
C00643=1060.503,352.262,-108.031,174.017,36.188,156.797
C00644=1060.496,352.014,-107.994,174.013,36.183,156.796
C00645=1060.490,351.767,-107.957,174.009,36.177,156.795
C00646=1060.483,351.520,-107.921,174.005,36.172,156.794
C00647=1060.475,351.273,-107.884,174.000,36.167,156.793
C00648=1060.468,351.026,-107.847,173.996,36.162,156.791
C00649=1060.462,350.779,-107.811,173.992,36.157,156.790
C00650=1060.455,350.531,-107.774,173.987,36.152,156.789
C00651=1060.448,350.284,-107.738,173.984,36.146,156.788
C00652=1060.441,350.037,-107.701,173.979,36.141,156.787
C00653=1060.434,349.790,-107.664,173.975,36.136,156.786
C00654=1060.427,349.542,-107.627,173.971,36.131,156.784
C00655=1060.420,349.295,-107.591,173.967,36.126,156.783
C00656=1060.414,349.048,-107.555,173.963,36.120,156.782
C00657=1060.407,348.801,-107.518,173.959,36.115,156.781
C00658=1060.400,348.554,-107.482,173.954,36.110,156.780
C00659=1060.393,348.306,-107.446,173.951,36.105,156.779
C00660=1060.387,348.059,-107.409,173.946,36.100,156.777
C00661=1060.380,347.812,-107.373,173.943,36.095,156.776
C00662=1060.373,347.565,-107.336,173.938,36.090,156.775
C00663=1060.366,347.317,-107.300,173.934,36.085,156.774
C00664=1060.360,347.070,-107.264,173.930,36.080,156.773
C00665=1060.353,346.826,-107.228,173.926,36.075,156.772
C00666=1060.346,346.583,-107.193,173.921,36.070,156.771
C00667=1060.340,346.340,-107.157,173.918,36.065,156.770
C00668=1060.333,346.097,-107.122,173.913,36.060,156.768
C00669=1060.326,345.853,-107.086,173.910,36.055,156.767
C00670=1060.319,345.610,-107.050,173.906,36.050,156.766
C00671=1060.313,345.367,-107.015,173.902,36.045,156.765
C00672=1060.307,345.123,-106.979,173.898,36.040,156.764
C00673=1060.300,344.876,-106.943,173.893,36.035,156.763
C00674=1060.293,344.629,-106.906,173.890,36.030,156.762
C00675=1060.286,344.381,-106.871,173.885,36.025,156.761
C00676=1060.280,344.134,-106.835,173.882,36.020,156.759
C00677=1060.273,343.888,-106.799,173.878,36.015,156.758
C00678=1060.266,343.639,-106.763,173.873,36.010,156.757
C00679=1060.260,343.392,-106.726,173.870,36.005,156.756
C00680=1060.253,343.145,-106.691,173.865,36.000,156.755
C00681=1060.246,342.898,-106.655,173.862,35.995,156.754
C00682=1060.239,342.650,-106.619,173.857,35.991,156.753
C00683=1060.232,342.403,-106.583,173.854,35.986,156.752
C00684=1060.226,342.155,-106.548,173.850,35.981,156.751
C00685=1060.219,341.908,-106.512,173.845,35.976,156.749
C00686=1060.213,341.661,-106.477,173.842,35.971,156.748
C00687=1060.206,341.413,-106.440,173.837,35.966,156.747
C00688=1060.199,341.166,-106.405,173.834,35.961,156.746
C00689=1060.192,340.919,-106.370,173.830,35.957,156.745
C00690=1060.186,340.672,-106.333,173.826,35.951,156.744
C00691=1060.179,340.424,-106.298,173.822,35.947,156.743
C00692=1060.172,340.177,-106.263,173.818,35.942,156.742
C00693=1060.165,339.929,-106.226,173.814,35.937,156.741
C00694=1060.158,339.682,-106.191,173.810,35.932,156.740
C00695=1060.152,339.434,-106.156,173.806,35.928,156.739
C00696=1060.146,339.187,-106.120,173.802,35.923,156.738
C00697=1060.139,338.940,-106.084,173.799,35.918,156.737
C00698=1060.132,338.693,-106.049,173.794,35.913,156.735
C00699=1060.126,338.445,-106.013,173.791,35.908,156.734
C00700=1060.119,338.198,-105.978,173.787,35.904,156.733
C00701=1060.112,337.950,-105.943,173.783,35.899,156.732
C00702=1060.106,337.702,-105.907,173.779,35.894,156.731
C00703=1060.099,337.455,-105.872,173.776,35.889,156.730
C00704=1060.092,337.208,-105.836,173.771,35.884,156.729
C00705=1060.086,336.961,-105.801,173.767,35.880,156.728
C00706=1060.080,336.713,-105.766,173.764,35.875,156.727
C00707=1060.072,336.465,-105.730,173.760,35.870,156.726
C00708=1060.065,336.218,-105.695,173.756,35.865,156.725
C00709=1060.059,335.971,-105.660,173.752,35.861,156.724
C00710=1060.052,335.723,-105.625,173.749,35.856,156.723
C00711=1060.045,335.475,-105.590,173.744,35.852,156.722
C00712=1060.039,335.228,-105.555,173.741,35.847,156.721
C00713=1060.032,334.980,-105.520,173.737,35.842,156.720
C00714=1060.025,334.733,-105.485,173.733,35.837,156.719
C00715=1060.019,334.485,-105.449,173.729,35.833,156.718
C00716=1060.012,334.238,-105.414,173.726,35.828,156.717
C00717=1060.006,333.991,-105.379,173.722,35.824,156.716
C00718=1060.000,333.743,-105.345,173.718,35.819,156.715
C00719=1059.993,333.496,-105.310,173.714,35.814,156.714
C00720=1059.986,333.249,-105.274,173.711,35.810,156.713
C00721=1059.979,333.003,-105.240,173.707,35.805,156.712
C00722=1059.973,332.757,-105.206,173.703,35.801,156.711
C00723=1059.966,332.511,-105.170,173.699,35.796,156.710
C00724=1059.960,332.266,-105.136,173.696,35.791,156.709
C00725=1059.953,332.021,-105.102,173.692,35.787,156.708
C00726=1059.947,331.775,-105.066,173.688,35.782,156.707
C00727=1059.940,331.530,-105.032,173.684,35.778,156.705
C00728=1059.930,331.146,-104.978,173.679,35.770,156.704
C00729=1059.920,330.761,-104.924,173.673,35.763,156.702
C00730=1059.914,330.514,-104.889,173.669,35.759,156.701
C00731=1059.907,330.266,-104.855,173.666,35.754,156.700
C00732=1059.900,330.019,-104.820,173.662,35.750,156.699
C00733=1059.893,329.771,-104.786,173.658,35.745,156.698
C00734=1059.887,329.524,-104.751,173.654,35.741,156.697
C00735=1059.879,329.276,-104.717,173.651,35.736,156.696
C00736=1059.873,329.029,-104.682,173.647,35.732,156.695
C00737=1059.866,328.781,-104.647,173.644,35.727,156.694
C00738=1059.859,328.534,-104.614,173.640,35.723,156.694
C00739=1059.853,328.286,-104.579,173.636,35.719,156.693
C00740=1059.846,328.038,-104.544,173.633,35.714,156.692
C00741=1059.839,327.791,-104.511,173.629,35.710,156.691
C00742=1059.832,327.543,-104.475,173.626,35.705,156.690
C00743=1059.826,327.296,-104.441,173.621,35.701,156.689
C00744=1059.819,327.048,-104.407,173.618,35.696,156.688
C00745=1059.813,326.800,-104.373,173.614,35.692,156.687
C00746=1059.805,326.553,-104.339,173.611,35.687,156.686
C00747=1059.799,326.305,-104.304,173.607,35.683,156.685
C00748=1059.793,326.058,-104.270,173.603,35.679,156.684
C00749=1059.786,325.810,-104.236,173.600,35.674,156.683
C00750=1059.779,325.562,-104.202,173.596,35.670,156.682
C00751=1059.773,325.316,-104.167,173.593,35.666,156.681
C00752=1059.766,325.068,-104.133,173.589,35.661,156.680
C00753=1059.759,324.820,-104.099,173.586,35.657,156.679
C00754=1059.752,324.572,-104.065,173.582,35.652,156.678
C00755=1059.746,324.325,-104.031,173.578,35.648,156.677
C00756=1059.740,324.077,-103.997,173.574,35.644,156.676
C00757=1059.733,323.829,-103.963,173.571,35.639,156.675
C00758=1059.727,323.582,-103.929,173.568,35.635,156.674
C00759=1059.720,323.335,-103.895,173.564,35.630,156.673
C00760=1059.714,323.087,-103.861,173.561,35.626,156.672
C00761=1059.707,322.839,-103.826,173.557,35.622,156.671
C00762=1059.700,322.592,-103.793,173.554,35.617,156.670
C00763=1059.694,322.344,-103.758,173.550,35.613,156.670
C00764=1059.687,322.097,-103.725,173.546,35.608,156.669
C00765=1059.681,321.849,-103.691,173.542,35.604,156.668
C00766=1059.674,321.602,-103.657,173.539,35.600,156.667
C00767=1059.668,321.354,-103.622,173.536,35.596,156.666
C00768=1059.661,321.107,-103.589,173.532,35.591,156.665
C00769=1059.655,320.858,-103.555,173.529,35.587,156.664
C00770=1059.649,320.611,-103.521,173.525,35.582,156.663
C00771=1059.642,320.363,-103.487,173.522,35.578,156.662
C00772=1059.636,320.116,-103.453,173.518,35.574,156.661
C00773=1059.629,319.868,-103.419,173.515,35.570,156.660
C00774=1059.623,319.620,-103.386,173.512,35.565,156.659
C00775=1059.616,319.373,-103.352,173.508,35.561,156.658
C00776=1059.610,319.125,-103.318,173.505,35.556,156.657
C00777=1059.604,318.911,-103.289,173.501,35.553,156.657
C00778=1059.598,318.697,-103.261,173.498,35.549,156.656
C00779=1059.593,318.484,-103.231,173.496,35.545,156.655
C00780=1059.587,318.269,-103.202,173.492,35.542,156.654
C00781=1059.582,318.055,-103.173,173.490,35.538,156.653
C00782=1059.577,317.841,-103.144,173.487,35.534,156.653
C00783=1059.571,317.626,-103.114,173.483,35.530,156.652
C00784=1059.565,317.413,-103.085,173.481,35.527,156.651
C00785=1059.560,317.165,-103.052,173.477,35.522,156.650
C00786=1059.552,316.917,-103.018,173.474,35.518,156.649
C00787=1059.547,316.670,-102.985,173.471,35.514,156.648
C00788=1059.540,316.423,-102.951,173.467,35.509,156.647
C00789=1059.534,316.175,-102.917,173.464,35.505,156.646
C00790=1059.528,315.927,-102.884,173.460,35.501,156.645
C00791=1059.522,315.680,-102.850,173.457,35.497,156.644
C00792=1059.515,315.431,-102.817,173.454,35.493,156.644
C00793=1059.509,315.184,-102.783,173.450,35.488,156.643
C00794=1059.503,314.937,-102.750,173.447,35.484,156.642
C00795=1059.496,314.689,-102.716,173.443,35.480,156.641
C00796=1059.490,314.441,-102.683,173.440,35.475,156.640
C00797=1059.484,314.193,-102.650,173.437,35.471,156.639
C00798=1059.477,313.945,-102.616,173.433,35.467,156.638
C00799=1059.471,313.698,-102.583,173.430,35.462,156.637
C00800=1059.464,313.451,-102.550,173.426,35.458,156.636
C00801=1059.457,313.203,-102.517,173.423,35.454,156.635
C00802=1059.451,312.955,-102.484,173.420,35.450,156.635
C00803=1059.445,312.707,-102.451,173.416,35.446,156.634
C00804=1059.438,312.460,-102.417,173.413,35.442,156.633
C00805=1059.431,312.212,-102.385,173.410,35.438,156.632
C00806=1059.425,311.965,-102.352,173.406,35.434,156.631
C00807=1059.418,311.716,-102.319,173.403,35.430,156.630
C00808=1059.412,311.469,-102.286,173.399,35.426,156.629
C00809=1059.405,311.221,-102.253,173.396,35.422,156.628
C00810=1059.398,310.973,-102.219,173.393,35.417,156.628
C00811=1059.392,310.726,-102.187,173.389,35.413,156.627
C00812=1059.386,310.478,-102.154,173.386,35.409,156.626
C00813=1059.379,310.230,-102.121,173.383,35.405,156.625
C00814=1059.372,309.982,-102.088,173.379,35.401,156.624
C00815=1059.365,309.735,-102.056,173.376,35.397,156.623
C00816=1059.359,309.487,-102.023,173.372,35.393,156.622
C00817=1059.352,309.239,-101.990,173.370,35.389,156.622
C00818=1059.346,308.992,-101.957,173.367,35.385,156.621
C00819=1059.340,308.744,-101.925,173.363,35.381,156.620
C00820=1059.333,308.496,-101.892,173.360,35.377,156.619
C00821=1059.327,308.248,-101.859,173.357,35.373,156.618
C00822=1059.320,308.000,-101.826,173.353,35.368,156.617
C00823=1059.314,307.753,-101.793,173.350,35.364,156.616
C00824=1059.307,307.506,-101.761,173.347,35.360,156.615
C00825=1059.301,307.258,-101.728,173.343,35.356,156.615
C00826=1059.294,307.010,-101.696,173.340,35.352,156.614
C00827=1059.287,306.762,-101.662,173.336,35.348,156.613
C00828=1059.281,306.514,-101.630,173.333,35.344,156.612
C00829=1059.275,306.266,-101.598,173.331,35.340,156.611
C00830=1059.269,306.019,-101.565,173.327,35.336,156.610
C00831=1059.263,305.771,-101.532,173.324,35.332,156.609
C00832=1059.256,305.524,-101.500,173.321,35.328,156.609
C00833=1059.250,305.277,-101.468,173.317,35.324,156.608
C00834=1059.243,305.031,-101.435,173.314,35.320,156.607
C00835=1059.236,304.784,-101.403,173.311,35.316,156.606
C00836=1059.230,304.537,-101.371,173.307,35.312,156.605
C00837=1059.224,304.291,-101.338,173.305,35.308,156.604
C00838=1059.218,304.044,-101.306,173.302,35.304,156.604
C00839=1059.211,303.798,-101.273,173.298,35.299,156.603
C00840=1059.205,303.552,-101.242,173.295,35.295,156.602
C00841=1059.198,303.304,-101.209,173.292,35.292,156.601
C00842=1059.192,303.056,-101.177,173.288,35.288,156.600
C00843=1059.186,302.808,-101.144,173.286,35.284,156.599
C00844=1059.179,302.561,-101.112,173.283,35.280,156.598
C00845=1059.173,302.313,-101.080,173.279,35.275,156.598
C00846=1059.167,302.065,-101.047,173.276,35.271,156.597
C00847=1059.161,301.817,-101.015,173.273,35.267,156.596
C00848=1059.155,301.569,-100.982,173.269,35.263,156.595
C00849=1059.148,301.321,-100.951,173.267,35.259,156.594
C00850=1059.142,301.074,-100.918,173.264,35.255,156.593
C00851=1059.136,300.826,-100.886,173.260,35.251,156.593
C00852=1059.129,300.578,-100.853,173.257,35.247,156.592
C00853=1059.124,300.330,-100.822,173.253,35.243,156.591
C00854=1059.117,300.083,-100.790,173.251,35.239,156.590
C00855=1059.111,299.835,-100.758,173.248,35.235,156.589
C00856=1059.105,299.587,-100.725,173.244,35.231,156.588
C00857=1059.099,299.339,-100.693,173.241,35.227,156.588
C00858=1059.092,299.092,-100.661,173.239,35.223,156.587
C00859=1059.086,298.844,-100.629,173.235,35.219,156.586
C00860=1059.080,298.595,-100.597,173.232,35.215,156.585
C00861=1059.073,298.348,-100.564,173.229,35.211,156.584
C00862=1059.068,298.100,-100.532,173.225,35.207,156.583
C00863=1059.061,297.853,-100.500,173.223,35.203,156.582
C00864=1059.055,297.605,-100.468,173.220,35.199,156.582
C00865=1059.049,297.357,-100.436,173.217,35.195,156.581
C00866=1059.042,297.109,-100.405,173.213,35.191,156.580
C00867=1059.036,296.861,-100.372,173.211,35.187,156.579
C00868=1059.031,296.614,-100.340,173.207,35.183,156.578
C00869=1059.024,296.366,-100.309,173.204,35.179,156.578
C00870=1059.018,296.117,-100.277,173.201,35.175,156.577
C00871=1059.011,295.870,-100.245,173.199,35.171,156.576
C00872=1059.005,295.622,-100.212,173.195,35.167,156.575
C00873=1058.998,295.374,-100.181,173.192,35.163,156.574
C00874=1058.992,295.126,-100.149,173.189,35.159,156.573
C00875=1058.985,294.878,-100.118,173.186,35.156,156.573
C00876=1058.979,294.631,-100.087,173.183,35.151,156.572
C00877=1058.973,294.383,-100.055,173.180,35.148,156.571
C00878=1058.967,294.135,-100.023,173.176,35.144,156.570
C00879=1058.961,293.886,-99.991,173.174,35.140,156.569
C00880=1058.954,293.639,-99.960,173.171,35.136,156.569
C00881=1058.947,293.391,-99.928,173.167,35.132,156.568
C00882=1058.942,293.143,-99.897,173.165,35.128,156.567
C00883=1058.935,292.895,-99.865,173.162,35.124,156.566
C00884=1058.928,292.647,-99.834,173.159,35.120,156.565
C00885=1058.922,292.399,-99.802,173.155,35.117,156.565
C00886=1058.916,292.151,-99.770,173.153,35.113,156.564
C00887=1058.909,291.904,-99.739,173.150,35.109,156.563
C00888=1058.903,291.656,-99.707,173.146,35.105,156.562
C00889=1058.896,291.417,-99.677,173.144,35.101,156.561
C00890=1058.891,291.179,-99.647,173.141,35.097,156.561
C00891=1058.885,290.940,-99.617,173.138,35.094,156.560
C00892=1058.878,290.701,-99.586,173.135,35.090,156.559
C00893=1058.873,290.462,-99.557,173.132,35.086,156.558
C00894=1058.867,290.223,-99.526,173.130,35.082,156.557
C00895=1058.860,289.984,-99.495,173.126,35.079,156.557
C00896=1058.855,289.746,-99.466,173.124,35.075,156.556
C00897=1058.848,289.498,-99.434,173.121,35.071,156.555
C00898=1058.842,289.250,-99.403,173.117,35.067,156.554
C00899=1058.835,289.001,-99.372,173.115,35.064,156.554
C00900=1058.829,288.754,-99.341,173.112,35.059,156.553
C00901=1058.823,288.506,-99.309,173.109,35.056,156.552
C00902=1058.816,288.258,-99.278,173.106,35.052,156.551
C00903=1058.811,288.010,-99.247,173.103,35.048,156.550
C00904=1058.804,287.762,-99.216,173.100,35.044,156.550
C00905=1058.797,287.514,-99.185,173.097,35.041,156.549
C00906=1058.791,287.267,-99.154,173.094,35.036,156.548
C00907=1058.785,287.019,-99.123,173.091,35.033,156.547
C00908=1058.778,286.770,-99.092,173.089,35.029,156.547
C00909=1058.771,286.522,-99.060,173.085,35.025,156.546
C00910=1058.766,286.274,-99.030,173.082,35.022,156.545
C00911=1058.759,286.027,-98.999,173.080,35.017,156.544
C00912=1058.753,285.779,-98.968,173.076,35.014,156.543
C00913=1058.746,285.531,-98.937,173.073,35.010,156.543
C00914=1058.740,285.282,-98.906,173.071,35.006,156.542
C00915=1058.734,285.035,-98.875,173.068,35.003,156.541
C00916=1058.727,284.787,-98.844,173.065,34.998,156.540
C00917=1058.721,284.538,-98.812,173.062,34.995,156.540
C00918=1058.716,284.291,-98.782,173.059,34.991,156.539
C00919=1058.709,284.043,-98.751,173.056,34.987,156.538
C00920=1058.703,283.795,-98.720,173.053,34.983,156.537
C00921=1058.697,283.546,-98.689,173.051,34.980,156.536
C00922=1058.690,283.298,-98.658,173.048,34.976,156.536
C00923=1058.684,283.051,-98.628,173.044,34.972,156.535
C00924=1058.678,282.802,-98.597,173.042,34.968,156.534
C00925=1058.672,282.555,-98.566,173.039,34.964,156.533
C00926=1058.665,282.306,-98.535,173.036,34.961,156.532
C00927=1058.659,282.058,-98.505,173.033,34.956,156.532
C00928=1058.653,281.811,-98.473,173.030,34.953,156.531
C00929=1058.647,281.563,-98.443,173.028,34.949,156.530
C00930=1058.640,281.315,-98.413,173.024,34.945,156.529
C00931=1058.633,281.067,-98.382,173.022,34.942,156.529
C00932=1058.627,280.819,-98.351,173.019,34.937,156.528
C00933=1058.621,280.571,-98.321,173.017,34.934,156.527
C00934=1058.615,280.322,-98.290,173.013,34.930,156.526
C00935=1058.609,280.075,-98.260,173.011,34.926,156.525
C00936=1058.602,279.827,-98.228,173.008,34.923,156.525
C00937=1058.596,279.579,-98.198,173.004,34.918,156.524
C00938=1058.590,279.330,-98.167,173.002,34.915,156.523
C00939=1058.584,279.083,-98.137,172.999,34.911,156.522
C00940=1058.577,278.834,-98.107,172.997,34.907,156.522
C00941=1058.571,278.587,-98.076,172.993,34.904,156.521
C00942=1058.565,278.338,-98.046,172.991,34.900,156.520
C00943=1058.559,278.090,-98.015,172.988,34.896,156.519
C00944=1058.552,277.842,-97.985,172.986,34.892,156.519
C00945=1058.546,277.609,-97.956,172.982,34.889,156.518
C00946=1058.540,277.376,-97.928,172.980,34.885,156.517
C00947=1058.534,277.142,-97.899,172.977,34.882,156.516
C00948=1058.529,276.909,-97.870,172.975,34.878,156.516
C00949=1058.523,276.675,-97.842,172.972,34.874,156.515
C00950=1058.517,276.442,-97.814,172.969,34.871,156.514
C00951=1058.511,276.209,-97.785,172.967,34.867,156.514
C00952=1058.505,275.975,-97.756,172.965,34.864,156.513
C00953=1058.498,275.728,-97.726,172.961,34.860,156.512
C00954=1058.492,275.480,-97.696,172.959,34.857,156.511
C00955=1058.486,275.231,-97.665,172.956,34.852,156.510
C00956=1058.480,274.983,-97.636,172.953,34.849,156.510
C00957=1058.473,274.735,-97.605,172.950,34.845,156.509
C00958=1058.468,274.487,-97.575,172.947,34.842,156.508
C00959=1058.461,274.239,-97.545,172.945,34.838,156.507
C00960=1058.455,273.991,-97.515,172.943,34.834,156.507
C00961=1058.449,273.743,-97.484,172.939,34.830,156.506
C00962=1058.442,273.494,-97.455,172.937,34.826,156.505
C00963=1058.436,273.246,-97.425,172.934,34.823,156.504
C00964=1058.430,272.998,-97.394,172.932,34.819,156.504
C00965=1058.423,272.750,-97.364,172.928,34.815,156.503
C00966=1058.418,272.502,-97.334,172.926,34.811,156.502
C00967=1058.411,272.254,-97.305,172.923,34.808,156.501
C00968=1058.405,272.006,-97.274,172.921,34.804,156.501
C00969=1058.398,271.758,-97.245,172.917,34.800,156.500
C00970=1058.393,271.510,-97.215,172.915,34.796,156.499
C00971=1058.385,271.262,-97.184,172.912,34.793,156.498
C00972=1058.380,271.013,-97.155,172.910,34.789,156.498
C00973=1058.373,270.766,-97.125,172.906,34.785,156.497
C00974=1058.367,270.517,-97.094,172.904,34.781,156.496
C00975=1058.361,270.269,-97.065,172.901,34.778,156.495
C00976=1058.355,270.021,-97.035,172.899,34.774,156.495
C00977=1058.348,269.772,-97.006,172.896,34.770,156.494
C00978=1058.342,269.524,-96.975,172.893,34.767,156.493
C00979=1058.336,269.276,-96.946,172.891,34.763,156.492
C00980=1058.330,269.029,-96.916,172.888,34.759,156.492
C00981=1058.323,268.780,-96.886,172.886,34.755,156.491
C00982=1058.317,268.532,-96.856,172.882,34.752,156.490
C00983=1058.311,268.284,-96.827,172.880,34.748,156.489
C00984=1058.305,268.036,-96.797,172.877,34.744,156.489
C00985=1058.299,267.787,-96.767,172.875,34.741,156.488
C00986=1058.292,267.540,-96.737,172.872,34.737,156.487
C00987=1058.286,267.291,-96.708,172.869,34.733,156.486
C00988=1058.279,267.043,-96.678,172.867,34.730,156.486
C00989=1058.273,266.795,-96.649,172.864,34.726,156.485
C00990=1058.267,266.547,-96.620,172.861,34.722,156.484
C00991=1058.261,266.299,-96.589,172.859,34.718,156.483
C00992=1058.255,266.051,-96.560,172.856,34.715,156.483
C00993=1058.248,265.802,-96.531,172.854,34.711,156.482
C00994=1058.242,265.554,-96.500,172.851,34.707,156.481
C00995=1058.236,265.306,-96.471,172.848,34.704,156.481
C00996=1058.230,265.058,-96.442,172.846,34.700,156.480
C00997=1058.224,264.810,-96.412,172.843,34.696,156.479
C00998=1058.217,264.561,-96.383,172.841,34.692,156.478
C00999=1058.211,264.313,-96.354,172.837,34.689,156.478
C01000=1058.204,264.065,-96.325,172.835,34.685,156.477
C01001=1058.199,263.834,-96.296,172.833,34.682,156.476
C01002=1058.193,263.603,-96.269,172.831,34.678,156.475
C01003=1058.187,263.370,-96.241,172.827,34.675,156.475
C01004=1058.182,263.139,-96.214,172.825,34.671,156.474
C01005=1058.176,262.908,-96.187,172.823,34.668,156.473
C01006=1058.170,262.677,-96.159,172.821,34.664,156.473
C01007=1058.163,262.445,-96.132,172.818,34.661,156.472
C01008=1058.157,262.214,-96.105,172.815,34.658,156.471
C01009=1058.151,261.966,-96.076,172.813,34.654,156.471
C01010=1058.145,261.718,-96.047,172.810,34.651,156.470
C01011=1058.138,261.469,-96.018,172.808,34.647,156.469
C01012=1058.132,261.221,-95.989,172.806,34.643,156.468
C01013=1058.125,260.973,-95.960,172.802,34.639,156.468
C01014=1058.119,260.725,-95.931,172.800,34.636,156.467
C01015=1058.113,260.476,-95.902,172.798,34.632,156.466
C01016=1058.107,260.228,-95.873,172.795,34.628,156.466
C01017=1058.100,259.979,-95.843,172.793,34.625,156.465
C01018=1058.094,259.731,-95.814,172.790,34.621,156.464
C01019=1058.087,259.483,-95.785,172.787,34.618,156.463
C01020=1058.081,259.235,-95.756,172.785,34.614,156.463
C01021=1058.075,258.987,-95.727,172.783,34.610,156.462
C01022=1058.069,258.739,-95.698,172.779,34.607,156.461
C01023=1058.062,258.491,-95.670,172.777,34.603,156.461
C01024=1058.055,258.243,-95.640,172.775,34.599,156.460
C01025=1058.049,257.994,-95.612,172.772,34.595,156.459
C01026=1058.043,257.745,-95.583,172.770,34.592,156.458
C01027=1058.036,257.497,-95.554,172.767,34.588,156.458
C01028=1058.030,257.249,-95.525,172.764,34.585,156.457
C01029=1058.024,257.001,-95.496,172.762,34.581,156.456
C01030=1058.018,256.753,-95.467,172.760,34.577,156.455
C01031=1058.012,256.504,-95.438,172.757,34.574,156.455
C01032=1058.005,256.256,-95.409,172.754,34.570,156.454
C01033=1057.999,256.008,-95.380,172.752,34.566,156.453
C01034=1057.993,255.760,-95.351,172.749,34.562,156.452
C01035=1057.986,255.512,-95.323,172.747,34.559,156.452
C01036=1057.980,255.263,-95.294,172.745,34.555,156.451
C01037=1057.974,255.015,-95.265,172.741,34.552,156.450
C01038=1057.967,254.767,-95.236,172.739,34.548,156.450
C01039=1057.961,254.518,-95.208,172.737,34.544,156.449
C01040=1057.955,254.270,-95.179,172.735,34.541,156.448
C01041=1057.949,254.022,-95.150,172.731,34.537,156.447
C01042=1057.943,253.774,-95.121,172.729,34.533,156.447
C01043=1057.937,253.525,-95.093,172.727,34.529,156.446
C01044=1057.930,253.277,-95.064,172.725,34.526,156.445
C01045=1057.924,253.028,-95.036,172.722,34.522,156.444
C01046=1057.918,252.780,-95.007,172.719,34.519,156.444
C01047=1057.911,252.532,-94.978,172.717,34.514,156.443
C01048=1057.905,252.283,-94.949,172.715,34.511,156.442
C01049=1057.899,252.035,-94.920,172.712,34.507,156.442
C01050=1057.894,251.787,-94.892,172.710,34.504,156.441
C01051=1057.887,251.539,-94.864,172.707,34.500,156.440
C01052=1057.881,251.291,-94.835,172.705,34.496,156.439
C01053=1057.875,251.042,-94.807,172.702,34.492,156.439
C01054=1057.868,250.794,-94.777,172.700,34.489,156.438
C01055=1057.862,250.545,-94.749,172.698,34.485,156.437
C01056=1057.856,250.297,-94.720,172.695,34.481,156.436
C01057=1057.851,250.065,-94.694,172.693,34.478,156.436
C01058=1057.845,249.833,-94.667,172.690,34.474,156.435
C01059=1057.839,249.600,-94.640,172.688,34.470,156.434
C01060=1057.834,249.368,-94.614,172.686,34.467,156.434
C01061=1057.828,249.135,-94.587,172.684,34.464,156.433
C01062=1057.822,248.903,-94.560,172.681,34.460,156.432
C01063=1057.816,248.671,-94.534,172.679,34.457,156.432
C01064=1057.810,248.438,-94.507,172.677,34.453,156.431
C01065=1057.804,248.189,-94.479,172.675,34.449,156.430
C01066=1057.798,247.942,-94.451,172.673,34.446,156.429
C01067=1057.792,247.693,-94.422,172.669,34.442,156.429
C01068=1057.786,247.445,-94.394,172.667,34.438,156.428
C01069=1057.780,247.197,-94.365,172.665,34.434,156.427
C01070=1057.774,246.948,-94.336,172.663,34.431,156.426
C01071=1057.768,246.700,-94.309,172.661,34.427,156.426
C01072=1057.762,246.452,-94.280,172.658,34.423,156.425
C01073=1057.756,246.203,-94.252,172.655,34.419,156.424
C01074=1057.750,245.954,-94.223,172.653,34.416,156.423
C01075=1057.743,245.706,-94.196,172.651,34.412,156.423
C01076=1057.737,245.459,-94.167,172.649,34.409,156.422
C01077=1057.731,245.210,-94.139,172.646,34.405,156.421
C01078=1057.725,244.961,-94.111,172.643,34.401,156.421
C01079=1057.719,244.713,-94.083,172.641,34.397,156.420
C01080=1057.712,244.464,-94.055,172.639,34.393,156.419
C01081=1057.707,244.216,-94.027,172.637,34.390,156.418
C01082=1057.700,243.968,-93.998,172.635,34.386,156.418
C01083=1057.694,243.720,-93.970,172.632,34.383,156.417
C01084=1057.687,243.471,-93.942,172.629,34.378,156.416
C01085=1057.682,243.223,-93.914,172.627,34.375,156.415
C01086=1057.675,242.975,-93.887,172.625,34.371,156.415
C01087=1057.669,242.726,-93.858,172.623,34.368,156.414
C01088=1057.663,242.477,-93.830,172.620,34.364,156.413
C01089=1057.657,242.229,-93.803,172.618,34.360,156.412
C01090=1057.651,241.981,-93.774,172.615,34.356,156.412
C01091=1057.645,241.732,-93.747,172.613,34.352,156.411
C01092=1057.638,241.484,-93.719,172.611,34.349,156.410
C01093=1057.633,241.236,-93.691,172.608,34.345,156.410
C01094=1057.626,240.987,-93.663,172.606,34.342,156.409
C01095=1057.619,240.739,-93.636,172.604,34.338,156.408
C01096=1057.613,240.490,-93.607,172.602,34.334,156.408
C01097=1057.607,240.242,-93.580,172.599,34.331,156.407
C01098=1057.600,239.994,-93.552,172.597,34.327,156.406
C01099=1057.595,239.745,-93.524,172.594,34.323,156.405
C01100=1057.588,239.497,-93.496,172.592,34.319,156.405
C01101=1057.582,239.249,-93.469,172.590,34.316,156.404
C01102=1057.576,239.000,-93.440,172.588,34.312,156.403
C01103=1057.569,238.752,-93.413,172.586,34.308,156.402
C01104=1057.563,238.504,-93.385,172.584,34.305,156.402
C01105=1057.557,238.255,-93.358,172.580,34.301,156.401
C01106=1057.551,238.006,-93.330,172.578,34.297,156.400
C01107=1057.545,237.758,-93.303,172.576,34.293,156.399
C01108=1057.538,237.510,-93.275,172.574,34.290,156.399
C01109=1057.531,237.262,-93.247,172.572,34.286,156.398
C01110=1057.526,237.013,-93.220,172.570,34.283,156.397
C01111=1057.520,236.764,-93.192,172.567,34.279,156.397
C01112=1057.513,236.516,-93.164,172.565,34.275,156.396
C01113=1057.508,236.281,-93.138,172.563,34.272,156.395
C01114=1057.501,236.045,-93.113,172.561,34.268,156.395
C01115=1057.496,235.809,-93.086,172.559,34.264,156.394
C01116=1057.490,235.575,-93.060,172.557,34.261,156.393
C01117=1057.484,235.339,-93.034,172.554,34.257,156.392
C01118=1057.478,235.103,-93.008,172.552,34.254,156.392
C01119=1057.473,234.868,-92.982,172.550,34.250,156.391
C01120=1057.466,234.633,-92.956,172.548,34.247,156.390
C01121=1057.461,234.384,-92.929,172.546,34.243,156.390
C01122=1057.454,234.136,-92.901,172.544,34.240,156.389
C01123=1057.448,233.887,-92.873,172.541,34.235,156.388
C01124=1057.442,233.639,-92.846,172.539,34.232,156.387
C01125=1057.435,233.390,-92.819,172.537,34.228,156.387
C01126=1057.430,233.142,-92.791,172.535,34.225,156.386
C01127=1057.423,232.893,-92.764,172.532,34.220,156.385
C01128=1057.417,232.646,-92.736,172.530,34.217,156.385
C01129=1057.411,232.397,-92.709,172.527,34.213,156.384
C01130=1057.404,232.148,-92.682,172.525,34.209,156.383
C01131=1057.398,231.900,-92.655,172.523,34.206,156.382
C01132=1057.392,231.651,-92.627,172.521,34.202,156.382
C01133=1057.386,231.403,-92.601,172.519,34.198,156.381
C01134=1057.379,231.154,-92.573,172.517,34.194,156.380
C01135=1057.374,230.906,-92.546,172.514,34.191,156.379
C01136=1057.368,230.657,-92.518,172.512,34.187,156.379
C01137=1057.362,230.409,-92.491,172.510,34.183,156.378
C01138=1057.355,230.161,-92.464,172.508,34.180,156.377
C01139=1057.349,229.912,-92.437,172.506,34.176,156.377
C01140=1057.343,229.664,-92.409,172.504,34.172,156.376
C01141=1057.337,229.415,-92.382,172.501,34.168,156.375
C01142=1057.331,229.166,-92.355,172.499,34.165,156.374
C01143=1057.324,228.919,-92.328,172.497,34.161,156.374
C01144=1057.318,228.670,-92.301,172.495,34.157,156.373
C01145=1057.312,228.421,-92.274,172.493,34.153,156.372
C01146=1057.305,228.173,-92.247,172.491,34.150,156.372
C01147=1057.299,227.924,-92.220,172.489,34.146,156.371
C01148=1057.293,227.676,-92.194,172.486,34.142,156.370
C01149=1057.286,227.427,-92.166,172.484,34.139,156.369
C01150=1057.280,227.179,-92.139,172.482,34.135,156.369
C01151=1057.275,226.930,-92.113,172.480,34.131,156.368
C01152=1057.268,226.682,-92.085,172.478,34.127,156.367
C01153=1057.261,226.434,-92.059,172.476,34.124,156.366
C01154=1057.255,226.185,-92.032,172.473,34.120,156.366
C01155=1057.249,225.937,-92.005,172.471,34.116,156.365
C01156=1057.243,225.688,-91.978,172.469,34.113,156.364
C01157=1057.237,225.440,-91.951,172.467,34.108,156.364
C01158=1057.230,225.191,-91.924,172.465,34.105,156.363
C01159=1057.224,224.943,-91.898,172.463,34.101,156.362
C01160=1057.217,224.694,-91.871,172.461,34.098,156.361
C01161=1057.212,224.445,-91.844,172.458,34.094,156.361
C01162=1057.206,224.198,-91.817,172.456,34.090,156.360
C01163=1057.199,223.948,-91.790,172.454,34.086,156.359
C01164=1057.193,223.700,-91.763,172.452,34.082,156.359
C01165=1057.186,223.451,-91.737,172.450,34.079,156.358
C01166=1057.181,223.203,-91.710,172.448,34.074,156.357
C01167=1057.175,222.955,-91.683,172.445,34.071,156.356
C01168=1057.168,222.706,-91.656,172.443,34.067,156.356
C01169=1057.162,222.467,-91.631,172.441,34.064,156.355
C01170=1057.157,222.227,-91.605,172.439,34.060,156.354
C01171=1057.150,221.988,-91.580,172.437,34.056,156.353
C01172=1057.145,221.748,-91.554,172.436,34.053,156.353
C01173=1057.139,221.509,-91.528,172.434,34.049,156.352
C01174=1057.133,221.269,-91.502,172.432,34.045,156.351
C01175=1057.127,221.030,-91.477,172.429,34.042,156.351
C01176=1057.122,220.791,-91.451,172.427,34.038,156.350
C01177=1057.114,220.542,-91.425,172.425,34.034,156.349
C01178=1057.109,220.294,-91.398,172.423,34.030,156.348
C01179=1057.102,220.046,-91.372,172.421,34.027,156.348
C01180=1057.096,219.797,-91.345,172.419,34.023,156.347
C01181=1057.089,219.549,-91.319,172.417,34.019,156.346
C01182=1057.083,219.300,-91.292,172.415,34.016,156.346
C01183=1057.077,219.051,-91.265,172.413,34.012,156.345
C01184=1057.071,218.803,-91.239,172.411,34.008,156.344
C01185=1057.064,218.554,-91.212,172.409,34.004,156.343
C01186=1057.058,218.306,-91.187,172.407,34.001,156.343
C01187=1057.052,218.057,-91.160,172.405,33.996,156.342
C01188=1057.045,217.808,-91.134,172.403,33.993,156.341
C01189=1057.039,217.560,-91.107,172.400,33.989,156.341
C01190=1057.033,217.312,-91.081,172.398,33.985,156.340
C01191=1057.027,217.064,-91.054,172.396,33.981,156.339
C01192=1057.020,216.814,-91.029,172.394,33.978,156.338
C01193=1057.015,216.566,-91.002,172.392,33.974,156.338
C01194=1057.009,216.318,-90.975,172.391,33.970,156.337
C01195=1057.002,216.069,-90.949,172.389,33.966,156.336
C01196=1056.996,215.820,-90.923,172.386,33.962,156.335
C01197=1056.990,215.572,-90.897,172.384,33.959,156.335
C01198=1056.984,215.323,-90.870,172.382,33.955,156.334
C01199=1056.977,215.075,-90.844,172.380,33.951,156.333
C01200=1056.971,214.826,-90.818,172.378,33.947,156.332
C01201=1056.965,214.578,-90.792,172.376,33.944,156.332
C01202=1056.959,214.329,-90.765,172.374,33.939,156.331
C01203=1056.953,214.081,-90.740,172.373,33.936,156.330
C01204=1056.946,213.832,-90.713,172.370,33.932,156.330
C01205=1056.940,213.584,-90.687,172.368,33.928,156.329
C01206=1056.934,213.335,-90.661,172.366,33.924,156.328
C01207=1056.928,213.087,-90.635,172.364,33.921,156.327
C01208=1056.922,212.838,-90.608,172.362,33.916,156.327
C01209=1056.915,212.589,-90.582,172.360,33.913,156.326
C01210=1056.910,212.340,-90.556,172.359,33.909,156.325
C01211=1056.903,212.092,-90.530,172.356,33.905,156.324
C01212=1056.897,211.844,-90.504,172.354,33.901,156.324
C01213=1056.891,211.595,-90.478,172.352,33.897,156.323
C01214=1056.884,211.346,-90.452,172.350,33.893,156.322
C01215=1056.878,211.098,-90.426,172.348,33.890,156.321
C01216=1056.872,210.849,-90.400,172.346,33.886,156.321
C01217=1056.866,210.601,-90.374,172.345,33.882,156.320
C01218=1056.860,210.352,-90.349,172.343,33.878,156.319
C01219=1056.854,210.104,-90.322,172.341,33.874,156.318
C01220=1056.847,209.855,-90.296,172.338,33.870,156.318
C01221=1056.841,209.606,-90.271,172.336,33.867,156.317
C01222=1056.834,209.358,-90.245,172.334,33.863,156.316
C01223=1056.829,209.109,-90.219,172.333,33.859,156.315
C01224=1056.822,208.861,-90.193,172.331,33.855,156.315
C01225=1056.816,208.624,-90.168,172.329,33.851,156.314
C01226=1056.810,208.388,-90.144,172.327,33.848,156.313
C01227=1056.804,208.150,-90.119,172.325,33.844,156.313
C01228=1056.798,207.913,-90.095,172.323,33.840,156.312
C01229=1056.792,207.676,-90.070,172.321,33.837,156.311
C01230=1056.786,207.440,-90.045,172.319,33.833,156.311
C01231=1056.781,207.203,-90.021,172.318,33.830,156.310
C01232=1056.775,206.966,-89.997,172.316,33.826,156.309
C01233=1056.749,205.916,-89.892,172.118,33.736,156.297
C01234=1056.743,205.667,-89.867,172.116,33.734,156.296
C01235=1056.737,205.418,-89.842,172.114,33.731,156.296
C01236=1056.732,205.170,-89.817,172.111,33.727,156.295
C01237=1056.726,204.921,-89.792,172.109,33.724,156.295
C01238=1056.720,204.672,-89.767,172.107,33.721,156.294
C01239=1056.714,204.424,-89.743,172.104,33.719,156.294
C01240=1056.707,204.175,-89.718,172.102,33.715,156.293
C01241=1056.702,203.927,-89.694,172.100,33.712,156.292
C01242=1056.696,203.677,-89.669,172.097,33.709,156.292
C01243=1056.690,203.429,-89.644,172.095,33.707,156.291
C01244=1056.685,203.180,-89.620,172.093,33.704,156.291
C01245=1056.678,202.931,-89.594,172.090,33.700,156.290
C01246=1056.673,202.683,-89.570,172.088,33.697,156.290
C01247=1056.667,202.433,-89.545,172.086,33.695,156.289
C01248=1056.660,202.185,-89.521,172.084,33.692,156.289
C01249=1056.655,201.937,-89.496,172.080,33.688,156.288
C01250=1056.649,201.688,-89.471,172.078,33.685,156.288
C01251=1056.644,201.439,-89.447,172.076,33.683,156.287
C01252=1056.637,201.190,-89.423,172.073,33.680,156.287
C01253=1056.631,200.941,-89.398,172.071,33.677,156.286
C01254=1056.625,200.693,-89.374,172.069,33.674,156.286
C01255=1056.619,200.444,-89.349,172.067,33.671,156.285
C01256=1056.612,200.195,-89.325,172.064,33.668,156.285
C01257=1056.607,199.947,-89.301,172.062,33.665,156.284
C01258=1056.601,199.698,-89.275,172.060,33.663,156.284
C01259=1056.595,199.450,-89.252,172.057,33.659,156.283
C01260=1056.589,199.200,-89.227,172.055,33.657,156.283
C01261=1056.582,198.951,-89.203,172.053,33.654,156.282
C01262=1056.577,198.703,-89.179,172.051,33.651,156.282
C01263=1056.570,198.454,-89.154,172.048,33.648,156.281
C01264=1056.564,198.206,-89.130,172.046,33.645,156.280
C01265=1056.559,197.956,-89.105,172.044,33.642,156.280
C01266=1056.553,197.708,-89.082,172.041,33.639,156.279
C01267=1056.547,197.459,-89.057,172.038,33.637,156.279
C01268=1056.541,197.211,-89.033,172.036,33.634,156.278
C01269=1056.535,196.961,-89.009,172.034,33.631,156.278
C01270=1056.529,196.713,-88.985,172.032,33.628,156.277
C01271=1056.522,196.464,-88.960,172.029,33.625,156.277
C01272=1056.516,196.216,-88.936,172.027,33.622,156.276
C01273=1056.511,195.967,-88.911,172.025,33.620,156.276
C01274=1056.505,195.719,-88.888,172.023,33.617,156.275
C01275=1056.499,195.469,-88.863,172.020,33.614,156.275
C01276=1056.493,195.221,-88.839,172.018,33.611,156.274
C01277=1056.487,194.972,-88.815,172.016,33.608,156.274
C01278=1056.481,194.723,-88.791,172.014,33.605,156.273
C01279=1056.475,194.474,-88.767,172.012,33.603,156.273
C01280=1056.469,194.226,-88.743,172.009,33.600,156.272
C01281=1056.463,193.977,-88.718,172.007,33.597,156.272
C01282=1056.457,193.728,-88.695,172.005,33.594,156.271
C01283=1056.451,193.479,-88.670,172.003,33.591,156.271
C01284=1056.445,193.231,-88.646,172.000,33.588,156.270
C01285=1056.440,192.982,-88.622,171.998,33.585,156.270
C01286=1056.433,192.733,-88.598,171.995,33.583,156.269
C01287=1056.428,192.484,-88.574,171.993,33.579,156.269
C01288=1056.421,192.235,-88.550,171.991,33.577,156.268
C01289=1056.416,191.986,-88.526,171.989,33.574,156.268
C01290=1056.410,191.738,-88.503,171.986,33.571,156.267
C01291=1056.404,191.489,-88.478,171.984,33.569,156.267
C01292=1056.398,191.241,-88.454,171.982,33.565,156.266
C01293=1056.392,190.991,-88.430,171.980,33.563,156.266
C01294=1056.386,190.707,-88.403,171.977,33.559,156.265
C01295=1056.379,190.424,-88.375,171.975,33.556,156.265
C01296=1056.372,190.139,-88.348,171.972,33.553,156.264
C01297=1056.366,189.855,-88.321,171.970,33.550,156.264
C01298=1056.360,189.607,-88.297,171.968,33.547,156.263
C01299=1056.354,189.358,-88.273,171.965,33.544,156.263
C01300=1056.348,189.109,-88.249,171.963,33.541,156.262
C01301=1056.343,188.861,-88.225,171.961,33.538,156.262
C01302=1056.336,188.611,-88.201,171.959,33.536,156.261
C01303=1056.330,188.363,-88.178,171.957,33.533,156.261
C01304=1056.325,188.114,-88.154,171.955,33.530,156.260
C01305=1056.318,187.865,-88.130,171.953,33.527,156.259
C01306=1056.313,187.616,-88.106,171.950,33.524,156.259
C01307=1056.307,187.368,-88.082,171.948,33.521,156.259
C01308=1056.302,187.119,-88.058,171.945,33.519,156.258
C01309=1056.296,186.870,-88.035,171.943,33.516,156.257
C01310=1056.290,186.622,-88.011,171.941,33.513,156.257
C01311=1056.284,186.373,-87.987,171.939,33.510,156.256
C01312=1056.279,186.124,-87.964,171.937,33.507,156.256
C01313=1056.273,185.875,-87.939,171.934,33.505,156.256
C01314=1056.267,185.626,-87.916,171.932,33.502,156.255
C01315=1056.262,185.377,-87.892,171.930,33.499,156.255
C01316=1056.256,185.129,-87.868,171.928,33.496,156.254
C01317=1056.249,184.879,-87.845,171.926,33.493,156.254
C01318=1056.244,184.631,-87.821,171.924,33.490,156.253
C01319=1056.238,184.382,-87.798,171.922,33.488,156.253
C01320=1056.232,184.134,-87.774,171.920,33.485,156.252
C01321=1056.226,183.884,-87.751,171.917,33.482,156.252
C01322=1056.220,183.636,-87.727,171.915,33.479,156.251
C01323=1056.214,183.387,-87.704,171.913,33.477,156.251
C01324=1056.208,183.138,-87.680,171.911,33.474,156.250
C01325=1056.202,182.889,-87.657,171.909,33.472,156.250
C01326=1056.196,182.641,-87.634,171.907,33.469,156.249
C01327=1056.189,182.391,-87.610,171.905,33.466,156.249
C01328=1056.184,182.142,-87.587,171.902,33.463,156.248
C01329=1056.178,181.894,-87.564,171.900,33.461,156.248
C01330=1056.171,181.644,-87.540,171.898,33.458,156.248
C01331=1056.165,181.396,-87.517,171.896,33.456,156.247
C01332=1056.159,181.147,-87.494,171.894,33.453,156.247
C01333=1056.153,180.899,-87.471,171.892,33.451,156.246
C01334=1056.146,180.650,-87.447,171.890,33.448,156.246
C01335=1056.141,180.401,-87.425,171.888,33.445,156.245
C01336=1056.135,180.152,-87.402,171.884,33.442,156.245
C01337=1056.129,179.904,-87.378,171.882,33.440,156.244
C01338=1056.123,179.654,-87.355,171.880,33.437,156.244
C01339=1056.117,179.405,-87.332,171.878,33.435,156.243
C01340=1056.111,179.157,-87.308,171.876,33.432,156.243
C01341=1056.105,178.908,-87.285,171.874,33.429,156.242
C01342=1056.098,178.659,-87.262,171.872,33.427,156.242
C01343=1056.092,178.410,-87.239,171.870,33.424,156.242
C01344=1056.086,178.161,-87.216,171.868,33.422,156.241
C01345=1056.081,177.912,-87.193,171.866,33.419,156.241
C01346=1056.075,177.664,-87.170,171.864,33.416,156.240
C01347=1056.069,177.414,-87.146,171.861,33.414,156.240
C01348=1056.063,177.165,-87.124,171.859,33.411,156.239
C01349=1056.057,176.917,-87.100,171.857,33.408,156.239
C01350=1056.050,176.668,-87.078,171.855,33.406,156.238
C01351=1056.045,176.419,-87.055,171.853,33.403,156.238
C01352=1056.039,176.170,-87.032,171.851,33.400,156.237
C01353=1056.032,175.921,-87.008,171.849,33.398,156.237
C01354=1056.027,175.672,-86.985,171.847,33.395,156.237
C01355=1056.021,175.424,-86.962,171.845,33.392,156.236
C01356=1056.015,175.175,-86.939,171.843,33.390,156.236
C01357=1056.009,174.926,-86.916,171.841,33.387,156.235
C01358=1056.002,174.641,-86.890,171.838,33.384,156.235
C01359=1055.995,174.358,-86.864,171.836,33.381,156.234
C01360=1055.989,174.073,-86.837,171.834,33.378,156.234
C01361=1055.982,173.789,-86.811,171.831,33.375,156.233
C01362=1055.976,173.540,-86.788,171.829,33.372,156.233
C01363=1055.970,173.290,-86.765,171.827,33.370,156.232
C01364=1055.963,173.042,-86.742,171.825,33.367,156.232
C01365=1055.958,172.793,-86.720,171.823,33.365,156.231
C01366=1055.952,172.544,-86.697,171.821,33.362,156.231
C01367=1055.946,172.295,-86.674,171.819,33.360,156.230
C01368=1055.940,172.046,-86.651,171.817,33.356,156.230
C01369=1055.935,171.797,-86.628,171.815,33.354,156.229
C01370=1055.928,171.549,-86.605,171.813,33.351,156.229
C01371=1055.922,171.300,-86.582,171.811,33.349,156.229
C01372=1055.917,171.051,-86.560,171.809,33.346,156.228
C01373=1055.911,170.802,-86.537,171.807,33.344,156.228
C01374=1055.905,170.553,-86.514,171.805,33.341,156.227
C01375=1055.899,170.305,-86.491,171.802,33.338,156.227
C01376=1055.893,170.056,-86.468,171.800,33.335,156.226
C01377=1055.887,169.807,-86.445,171.798,33.333,156.226
C01378=1055.882,169.557,-86.423,171.796,33.330,156.225
C01379=1055.876,169.308,-86.400,171.794,33.328,156.225
C01380=1055.870,169.060,-86.378,171.792,33.325,156.224
C01381=1055.864,168.811,-86.355,171.790,33.323,156.224
C01382=1055.858,168.562,-86.332,171.788,33.320,156.224
C01383=1055.853,168.313,-86.309,171.786,33.317,156.223
C01384=1055.847,168.064,-86.286,171.784,33.314,156.223
C01385=1055.840,167.816,-86.264,171.782,33.312,156.222
C01386=1055.835,167.566,-86.241,171.780,33.309,156.222
C01387=1055.829,167.317,-86.219,171.778,33.307,156.221
C01388=1055.823,167.068,-86.196,171.776,33.304,156.221
C01389=1055.817,166.820,-86.173,171.774,33.302,156.220
C01390=1055.811,166.571,-86.150,171.772,33.299,156.220
C01391=1055.806,166.321,-86.128,171.770,33.296,156.219
C01392=1055.800,166.073,-86.105,171.768,33.293,156.219
C01393=1055.794,165.824,-86.083,171.766,33.291,156.219
C01394=1055.788,165.576,-86.060,171.764,33.288,156.218
C01395=1055.783,165.326,-86.038,171.762,33.286,156.218
C01396=1055.777,165.077,-86.015,171.760,33.283,156.217
C01397=1055.771,164.829,-85.993,171.758,33.281,156.217
C01398=1055.765,164.580,-85.970,171.756,33.278,156.216
C01399=1055.760,164.330,-85.947,171.754,33.275,156.216
C01400=1055.754,164.081,-85.925,171.752,33.272,156.215
C01401=1055.748,163.833,-85.902,171.750,33.270,156.215
C01402=1055.742,163.583,-85.880,171.748,33.267,156.214
C01403=1055.737,163.335,-85.857,171.746,33.265,156.214
C01404=1055.731,163.086,-85.834,171.744,33.262,156.214
C01405=1055.725,162.837,-85.813,171.742,33.259,156.213
C01406=1055.719,162.588,-85.790,171.740,33.257,156.213
C01407=1055.714,162.339,-85.767,171.739,33.254,156.212
C01408=1055.708,162.090,-85.745,171.737,33.251,156.212
C01409=1055.702,161.842,-85.723,171.735,33.249,156.211
C01410=1055.697,161.592,-85.700,171.733,33.246,156.211
C01411=1055.691,161.343,-85.678,171.731,33.244,156.210
C01412=1055.685,161.095,-85.655,171.729,33.241,156.210
C01413=1055.679,160.845,-85.633,171.727,33.238,156.210
C01414=1055.674,160.596,-85.610,171.725,33.236,156.209
C01415=1055.667,160.347,-85.588,171.723,33.233,156.209
C01416=1055.661,160.099,-85.566,171.721,33.231,156.208
C01417=1055.656,159.850,-85.544,171.719,33.228,156.208
C01418=1055.650,159.601,-85.522,171.717,33.226,156.207
C01419=1055.643,159.352,-85.500,171.715,33.223,156.207
C01420=1055.638,159.103,-85.477,171.713,33.220,156.206
C01421=1055.632,158.854,-85.456,171.711,33.218,156.206
C01422=1055.625,158.569,-85.430,171.709,33.215,156.206
C01423=1055.618,158.284,-85.405,171.707,33.212,156.205
C01424=1055.611,158.000,-85.379,171.705,33.210,156.205
C01425=1055.605,157.715,-85.354,171.702,33.206,156.204
C01426=1055.598,157.466,-85.333,171.701,33.204,156.204
C01427=1055.592,157.217,-85.310,171.699,33.201,156.203
C01428=1055.587,156.968,-85.288,171.697,33.199,156.203
C01429=1055.581,156.720,-85.266,171.695,33.197,156.202
C01430=1055.575,156.470,-85.244,171.693,33.194,156.202
C01431=1055.569,156.221,-85.222,171.691,33.192,156.202
C01432=1055.563,155.972,-85.200,171.689,33.189,156.201
C01433=1055.558,155.724,-85.178,171.687,33.187,156.201
C01434=1055.552,155.474,-85.156,171.685,33.184,156.200
C01435=1055.545,155.226,-85.134,171.683,33.181,156.200
C01436=1055.539,154.977,-85.112,171.681,33.179,156.199
C01437=1055.534,154.727,-85.090,171.679,33.176,156.199
C01438=1055.528,154.479,-85.069,171.677,33.174,156.198
C01439=1055.522,154.230,-85.047,171.676,33.171,156.198
C01440=1055.515,153.981,-85.025,171.674,33.169,156.198
C01441=1055.510,153.731,-85.003,171.672,33.167,156.197
C01442=1055.504,153.482,-84.981,171.670,33.164,156.197
C01443=1055.498,153.234,-84.959,171.668,33.161,156.196
C01444=1055.492,152.985,-84.937,171.666,33.159,156.196
C01445=1055.486,152.736,-84.916,171.664,33.156,156.196
C01446=1055.480,152.486,-84.894,171.662,33.154,156.195
C01447=1055.475,152.238,-84.872,171.660,33.152,156.195
C01448=1055.468,151.989,-84.850,171.658,33.149,156.194
C01449=1055.462,151.740,-84.828,171.656,33.147,156.194
C01450=1055.456,151.491,-84.807,171.655,33.144,156.193
C01451=1055.450,151.242,-84.785,171.653,33.142,156.193
C01452=1055.445,150.993,-84.763,171.651,33.139,156.193
C01453=1055.439,150.743,-84.742,171.649,33.136,156.192
C01454=1055.432,150.495,-84.719,171.647,33.134,156.192
C01455=1055.427,150.246,-84.698,171.645,33.132,156.191
C01456=1055.420,149.997,-84.676,171.643,33.129,156.191
C01457=1055.414,149.748,-84.655,171.641,33.127,156.191
C01458=1055.410,149.499,-84.633,171.640,33.124,156.190
C01459=1055.403,149.250,-84.611,171.638,33.122,156.190
C01460=1055.397,149.001,-84.589,171.636,33.119,156.189
C01461=1055.391,148.752,-84.568,171.634,33.117,156.189
C01462=1055.385,148.503,-84.547,171.632,33.115,156.188
C01463=1055.379,148.254,-84.525,171.630,33.112,156.188
C01464=1055.373,148.005,-84.503,171.628,33.109,156.188
C01465=1055.368,147.756,-84.482,171.626,33.107,156.187
C01466=1055.361,147.507,-84.460,171.625,33.104,156.187
C01467=1055.355,147.258,-84.439,171.623,33.102,156.186
C01468=1055.350,147.009,-84.418,171.621,33.100,156.186
C01469=1055.344,146.760,-84.396,171.619,33.097,156.186
C01470=1055.337,146.511,-84.374,171.617,33.095,156.185
C01471=1055.331,146.262,-84.353,171.615,33.092,156.185
C01472=1055.326,146.013,-84.331,171.613,33.089,156.184
C01473=1055.319,145.764,-84.310,171.611,33.087,156.184
C01474=1055.313,145.515,-84.288,171.610,33.085,156.183
C01475=1055.308,145.266,-84.267,171.608,33.082,156.183
C01476=1055.302,145.017,-84.245,171.606,33.080,156.183
C01477=1055.296,144.767,-84.224,171.604,33.078,156.182
C01478=1055.290,144.519,-84.203,171.602,33.075,156.182
C01479=1055.284,144.269,-84.181,171.600,33.073,156.181
C01480=1055.278,144.021,-84.161,171.598,33.070,156.181
C01481=1055.272,143.772,-84.139,171.597,33.068,156.181
C01482=1055.265,143.523,-84.117,171.595,33.066,156.180
C01483=1055.260,143.274,-84.096,171.593,33.063,156.180
C01484=1055.254,143.024,-84.075,171.591,33.060,156.179
C01485=1055.248,142.775,-84.054,171.589,33.058,156.179
C01486=1055.242,142.491,-84.029,171.587,33.055,156.178
C01487=1055.235,142.206,-84.005,171.585,33.053,156.178
C01488=1055.227,141.921,-83.981,171.583,33.050,156.177
C01489=1055.221,141.636,-83.956,171.581,33.047,156.177
C01490=1055.215,141.386,-83.934,171.579,33.044,156.177
C01491=1055.210,141.137,-83.914,171.577,33.042,156.176
C01492=1055.203,140.888,-83.892,171.575,33.040,156.176
C01493=1055.198,140.640,-83.871,171.573,33.037,156.175
C01494=1055.191,140.391,-83.850,171.572,33.035,156.175
C01495=1055.185,140.141,-83.829,171.570,33.032,156.175
C01496=1055.179,139.892,-83.808,171.568,33.030,156.174
C01497=1055.173,139.643,-83.786,171.566,33.028,156.174
C01498=1055.168,139.394,-83.765,171.564,33.025,156.173
C01499=1055.161,139.145,-83.744,171.562,33.022,156.173
C01500=1055.155,138.896,-83.723,171.561,33.020,156.173
C01501=1055.150,138.647,-83.702,171.559,33.018,156.172
C01502=1055.144,138.398,-83.681,171.557,33.015,156.172
C01503=1055.137,138.149,-83.660,171.555,33.013,156.171
C01504=1055.131,137.900,-83.639,171.553,33.010,156.171
C01505=1055.126,137.651,-83.618,171.552,33.008,156.171
C01506=1055.120,137.402,-83.596,171.550,33.006,156.170
C01507=1055.114,137.153,-83.576,171.548,33.003,156.170
C01508=1055.108,136.904,-83.555,171.546,33.001,156.169
C01509=1055.102,136.655,-83.534,171.544,32.998,156.169
C01510=1055.095,136.406,-83.513,171.542,32.996,156.169
C01511=1055.089,136.157,-83.491,171.541,32.993,156.168
C01512=1055.084,135.908,-83.471,171.539,32.991,156.168
C01513=1055.077,135.659,-83.450,171.537,32.989,156.167
C01514=1055.072,135.410,-83.429,171.535,32.986,156.167
C01515=1055.066,135.160,-83.407,171.533,32.984,156.167
C01516=1055.060,134.912,-83.388,171.532,32.982,156.166
C01517=1055.053,134.662,-83.366,171.530,32.979,156.166
C01518=1055.048,134.413,-83.345,171.528,32.977,156.165
C01519=1055.041,134.164,-83.324,171.526,32.975,156.165
C01520=1055.036,133.915,-83.304,171.524,32.972,156.165
C01521=1055.030,133.666,-83.282,171.523,32.970,156.164
C01522=1055.024,133.417,-83.262,171.521,32.968,156.164
C01523=1055.018,133.168,-83.241,171.519,32.965,156.163
C01524=1055.012,132.919,-83.220,171.517,32.962,156.163
C01525=1055.006,132.670,-83.200,171.515,32.960,156.162
C01526=1055.000,132.421,-83.178,171.514,32.958,156.162
C01527=1054.994,132.172,-83.158,171.512,32.955,156.162
C01528=1054.988,131.923,-83.137,171.510,32.953,156.161
C01529=1054.983,131.674,-83.116,171.508,32.950,156.161
C01530=1054.976,131.425,-83.095,171.506,32.948,156.161
C01531=1054.971,131.176,-83.075,171.505,32.946,156.160
C01532=1054.964,130.926,-83.054,171.503,32.944,156.160
C01533=1054.958,130.678,-83.034,171.501,32.941,156.159
C01534=1054.952,130.428,-83.013,171.499,32.938,156.159
C01535=1054.946,130.179,-82.993,171.497,32.936,156.159
C01536=1054.939,129.930,-82.972,171.496,32.934,156.158
C01537=1054.934,129.681,-82.951,171.494,32.932,156.158
C01538=1054.927,129.432,-82.931,171.492,32.929,156.157
C01539=1054.922,129.183,-82.910,171.490,32.927,156.157
C01540=1054.915,128.934,-82.889,171.488,32.925,156.157
C01541=1054.909,128.685,-82.869,171.487,32.922,156.156
C01542=1054.903,128.435,-82.848,171.485,32.920,156.156
C01543=1054.897,128.186,-82.828,171.483,32.918,156.155
C01544=1054.891,127.938,-82.808,171.481,32.916,156.155
C01545=1054.885,127.688,-82.787,171.480,32.913,156.155
C01546=1054.879,127.439,-82.767,171.478,32.911,156.154
C01547=1054.873,127.190,-82.747,171.476,32.909,156.154
C01548=1054.867,126.941,-82.725,171.474,32.906,156.154
C01549=1054.860,126.692,-82.705,171.472,32.903,156.153
C01550=1054.854,126.407,-82.682,171.471,32.901,156.153
C01551=1054.847,126.122,-82.658,171.469,32.898,156.152
C01552=1054.840,125.836,-82.635,171.467,32.896,156.152
C01553=1054.833,125.551,-82.612,171.465,32.893,156.151
C01554=1054.827,125.302,-82.591,171.464,32.890,156.151
C01555=1054.821,125.053,-82.571,171.462,32.888,156.151
C01556=1054.814,124.804,-82.550,171.460,32.886,156.150
C01557=1054.809,124.555,-82.530,171.458,32.883,156.150
C01558=1054.803,124.306,-82.510,171.457,32.881,156.149
C01559=1054.796,124.056,-82.490,171.455,32.879,156.149
C01560=1054.791,123.807,-82.469,171.453,32.877,156.149
C01561=1054.785,123.559,-82.449,171.451,32.874,156.148
C01562=1054.779,123.309,-82.429,171.450,32.872,156.148
C01563=1054.773,123.061,-82.407,171.448,32.870,156.148
C01564=1054.767,122.812,-82.388,171.446,32.867,156.147
C01565=1054.760,122.562,-82.367,171.444,32.864,156.147
C01566=1054.754,122.313,-82.347,171.442,32.862,156.146
C01567=1054.749,122.064,-82.327,171.441,32.860,156.146
C01568=1054.743,121.815,-82.306,171.439,32.857,156.146
C01569=1054.737,121.566,-82.286,171.437,32.855,156.145
C01570=1054.731,121.317,-82.266,171.436,32.853,156.145
C01571=1054.725,121.067,-82.246,171.434,32.851,156.144
C01572=1054.719,120.818,-82.226,171.432,32.848,156.144
C01573=1054.714,120.569,-82.205,171.430,32.846,156.144
C01574=1054.707,120.320,-82.185,171.429,32.844,156.143
C01575=1054.701,120.071,-82.165,171.427,32.841,156.143
C01576=1054.695,119.822,-82.145,171.425,32.839,156.142
C01577=1054.690,119.573,-82.124,171.423,32.837,156.142
C01578=1054.683,119.324,-82.104,171.422,32.834,156.142
C01579=1054.677,119.075,-82.084,171.420,32.831,156.141
C01580=1054.671,118.826,-82.064,171.418,32.829,156.141
C01581=1054.666,118.577,-82.043,171.416,32.827,156.140
C01582=1054.659,118.327,-82.023,171.415,32.824,156.140
C01583=1054.654,118.078,-82.004,171.413,32.822,156.140
C01584=1054.648,117.829,-81.983,171.411,32.820,156.139
C01585=1054.642,117.580,-81.963,171.410,32.817,156.139
C01586=1054.636,117.330,-81.943,171.408,32.815,156.139
C01587=1054.630,117.082,-81.923,171.406,32.813,156.138
C01588=1054.624,116.832,-81.902,171.404,32.810,156.138
C01589=1054.619,116.584,-81.883,171.403,32.808,156.137
C01590=1054.613,116.335,-81.863,171.401,32.805,156.137
C01591=1054.606,116.085,-81.843,171.399,32.803,156.137
C01592=1054.601,115.836,-81.822,171.398,32.800,156.136
C01593=1054.595,115.587,-81.802,171.396,32.798,156.136
C01594=1054.589,115.338,-81.782,171.394,32.796,156.135
C01595=1054.583,115.089,-81.763,171.393,32.793,156.135
C01596=1054.576,114.840,-81.742,171.392,32.791,156.135
C01597=1054.571,114.590,-81.722,171.390,32.789,156.134
C01598=1054.565,114.341,-81.702,171.388,32.786,156.134
C01599=1054.559,114.092,-81.682,171.387,32.784,156.133
C01600=1054.553,113.843,-81.663,171.385,32.781,156.133
C01601=1054.547,113.593,-81.643,171.383,32.779,156.133
C01602=1054.541,113.345,-81.623,171.381,32.777,156.132
C01603=1054.535,113.096,-81.603,171.380,32.774,156.132
C01604=1054.529,112.847,-81.583,171.378,32.772,156.131
C01605=1054.523,112.597,-81.564,171.376,32.770,156.131
C01606=1054.517,112.348,-81.543,171.375,32.768,156.131
C01607=1054.511,112.099,-81.523,171.373,32.765,156.130
C01608=1054.505,111.850,-81.504,171.371,32.763,156.130
C01609=1054.499,111.601,-81.484,171.369,32.761,156.130
C01610=1054.493,111.352,-81.464,171.368,32.758,156.129
C01611=1054.487,111.102,-81.445,171.366,32.756,156.129
C01612=1054.481,110.853,-81.425,171.364,32.753,156.128
C01613=1054.475,110.604,-81.405,171.363,32.752,156.128
C01614=1054.469,110.357,-81.386,171.361,32.749,156.128
C01615=1054.463,110.110,-81.366,171.359,32.747,156.127
C01616=1054.457,109.863,-81.346,171.357,32.744,156.127
C01617=1054.451,109.615,-81.326,171.356,32.742,156.127
C01618=1054.445,109.368,-81.308,171.354,32.740,156.126
C01619=1054.439,109.121,-81.288,171.352,32.738,156.126
C01620=1054.432,108.874,-81.268,171.351,32.735,156.125
C01621=1054.427,108.627,-81.250,171.349,32.733,156.125
C01622=1054.421,108.378,-81.230,171.347,32.731,156.125
C01623=1054.415,108.128,-81.210,171.346,32.729,156.124
C01624=1054.409,107.879,-81.190,171.344,32.726,156.124
C01625=1054.403,107.630,-81.171,171.342,32.724,156.124
C01626=1054.397,107.381,-81.151,171.340,32.721,156.123
C01627=1054.390,107.132,-81.132,171.339,32.720,156.123
C01628=1054.384,106.883,-81.112,171.337,32.717,156.122
C01629=1054.379,106.634,-81.093,171.336,32.714,156.122
C01630=1054.373,106.385,-81.073,171.335,32.712,156.122
C01631=1054.367,106.135,-81.054,171.333,32.710,156.121
C01632=1054.360,105.886,-81.034,171.331,32.708,156.121
C01633=1054.354,105.637,-81.015,171.330,32.705,156.120
C01634=1054.348,105.388,-80.995,171.328,32.703,156.120
C01635=1054.342,105.139,-80.976,171.326,32.701,156.120
C01636=1054.336,104.890,-80.956,171.324,32.699,156.119
C01637=1054.331,104.640,-80.937,171.323,32.696,156.119
C01638=1054.324,104.392,-80.917,171.321,32.694,156.119
C01639=1054.318,104.142,-80.898,171.319,32.691,156.118
C01640=1054.313,103.893,-80.879,171.318,32.689,156.118
C01641=1054.307,103.644,-80.859,171.316,32.687,156.118
C01642=1054.299,103.354,-80.837,171.314,32.684,156.117
C01643=1054.293,103.065,-80.814,171.312,32.682,156.117
C01644=1054.285,102.775,-80.791,171.310,32.679,156.116
C01645=1054.278,102.486,-80.769,171.308,32.676,156.116
C01646=1054.272,102.237,-80.749,171.307,32.674,156.115
C01647=1054.267,101.988,-80.730,171.305,32.671,156.115
C01648=1054.261,101.739,-80.710,171.303,32.669,156.115
C01649=1054.254,101.490,-80.692,171.301,32.667,156.114
C01650=1054.249,101.240,-80.672,171.300,32.664,156.114
C01651=1054.243,100.991,-80.653,171.298,32.662,156.113
C01652=1054.237,100.742,-80.633,171.296,32.660,156.113
C01653=1054.231,100.493,-80.614,171.295,32.658,156.113
C01654=1054.225,100.244,-80.595,171.293,32.655,156.112
C01655=1054.218,99.994,-80.577,171.291,32.653,156.112
C01656=1054.212,99.745,-80.556,171.290,32.650,156.112
C01657=1054.206,99.496,-80.537,171.289,32.648,156.111
C01658=1054.200,99.246,-80.518,171.287,32.646,156.111
C01659=1054.194,98.997,-80.499,171.286,32.644,156.111
C01660=1054.187,98.748,-80.480,171.284,32.641,156.110
C01661=1054.182,98.499,-80.460,171.282,32.639,156.110
C01662=1054.175,98.250,-80.442,171.281,32.637,156.109
C01663=1054.169,98.000,-80.423,171.279,32.635,156.109
C01664=1054.163,97.751,-80.404,171.277,32.633,156.109
C01665=1054.157,97.503,-80.384,171.276,32.630,156.108
C01666=1054.151,97.253,-80.365,171.274,32.628,156.108
C01667=1054.145,97.004,-80.346,171.272,32.626,156.108
C01668=1054.139,96.755,-80.327,171.271,32.624,156.107
C01669=1054.133,96.505,-80.308,171.269,32.621,156.107
C01670=1054.127,96.256,-80.289,171.267,32.619,156.106
C01671=1054.121,96.007,-80.270,171.265,32.616,156.106
C01672=1054.115,95.757,-80.251,171.264,32.614,156.106
C01673=1054.108,95.509,-80.232,171.262,32.612,156.105
C01674=1054.103,95.260,-80.212,171.260,32.610,156.105
C01675=1054.096,95.010,-80.194,171.259,32.607,156.105
C01676=1054.090,94.761,-80.175,171.257,32.605,156.104
C01677=1054.084,94.512,-80.156,171.255,32.603,156.104
C01678=1054.077,94.227,-80.134,171.254,32.600,156.103
C01679=1054.071,93.941,-80.113,171.252,32.598,156.103
C01680=1054.064,93.656,-80.091,171.250,32.595,156.103
C01681=1054.057,93.371,-80.069,171.248,32.592,156.102
C01682=1054.051,93.122,-80.050,171.247,32.590,156.102
C01683=1054.045,92.873,-80.031,171.246,32.588,156.101
C01684=1054.038,92.624,-80.012,171.244,32.586,156.101
C01685=1054.033,92.374,-79.993,171.242,32.583,156.101
C01686=1054.026,92.125,-79.974,171.241,32.581,156.100
C01687=1054.021,91.876,-79.955,171.239,32.579,156.100
C01688=1054.014,91.626,-79.936,171.237,32.576,156.100
C01689=1054.009,91.377,-79.917,171.236,32.574,156.099
C01690=1054.003,91.128,-79.900,171.234,32.571,156.099
C01691=1053.997,90.879,-79.880,171.232,32.569,156.098
C01692=1053.991,90.629,-79.862,171.231,32.567,156.098
C01693=1053.985,90.380,-79.842,171.229,32.565,156.098
C01694=1053.979,90.131,-79.824,171.227,32.563,156.097
C01695=1053.972,89.882,-79.805,171.226,32.560,156.097
C01696=1053.966,89.633,-79.786,171.224,32.558,156.097
C01697=1053.960,89.383,-79.767,171.222,32.556,156.096
C01698=1053.954,89.134,-79.749,171.221,32.554,156.096
C01699=1053.947,88.885,-79.730,171.219,32.552,156.096
C01700=1053.941,88.635,-79.712,171.217,32.549,156.095
C01701=1053.936,88.386,-79.693,171.216,32.547,156.095
C01702=1053.929,88.137,-79.674,171.214,32.544,156.094
C01703=1053.923,87.888,-79.656,171.212,32.542,156.094
C01704=1053.917,87.639,-79.637,171.211,32.540,156.094
C01705=1053.911,87.390,-79.618,171.210,32.538,156.093
C01706=1053.905,87.140,-79.600,171.208,32.536,156.093
C01707=1053.899,86.891,-79.581,171.207,32.533,156.093
C01708=1053.892,86.642,-79.563,171.205,32.531,156.092
C01709=1053.887,86.392,-79.543,171.203,32.529,156.092
C01710=1053.880,86.143,-79.525,171.202,32.527,156.092
C01711=1053.875,85.894,-79.507,171.200,32.525,156.091
C01712=1053.868,85.645,-79.489,171.198,32.522,156.091
C01713=1053.862,85.396,-79.470,171.197,32.520,156.091
C01714=1053.856,85.146,-79.451,171.195,32.517,156.090
C01715=1053.850,84.897,-79.433,171.193,32.515,156.090
C01716=1053.844,84.648,-79.414,171.192,32.513,156.089
C01717=1053.838,84.399,-79.396,171.190,32.511,156.089
C01718=1053.832,84.150,-79.377,171.188,32.509,156.089
C01719=1053.826,83.900,-79.359,171.187,32.506,156.088
C01720=1053.819,83.651,-79.340,171.185,32.504,156.088
C01721=1053.813,83.402,-79.321,171.183,32.502,156.088
C01722=1053.807,83.152,-79.303,171.182,32.500,156.087
C01723=1053.802,82.903,-79.285,171.180,32.497,156.087
C01724=1053.795,82.654,-79.266,171.178,32.495,156.087
C01725=1053.789,82.404,-79.248,171.177,32.493,156.086
C01726=1053.783,82.155,-79.229,171.176,32.491,156.086
C01727=1053.776,81.906,-79.211,171.174,32.488,156.085
C01728=1053.772,81.657,-79.193,171.173,32.486,156.085
C01729=1053.765,81.408,-79.174,171.171,32.484,156.085
C01730=1053.759,81.159,-79.155,171.169,32.481,156.084
C01731=1053.753,80.909,-79.137,171.168,32.479,156.084
C01732=1053.747,80.660,-79.119,171.166,32.477,156.084
C01733=1053.741,80.411,-79.101,171.165,32.475,156.083
C01734=1053.735,80.161,-79.082,171.163,32.472,156.083
C01735=1053.729,79.912,-79.063,171.161,32.470,156.083
C01736=1053.723,79.663,-79.046,171.160,32.468,156.082
C01737=1053.717,79.414,-79.027,171.158,32.466,156.082
C01738=1053.711,79.164,-79.009,171.156,32.463,156.081
C01739=1053.704,78.915,-78.990,171.155,32.461,156.081
C01740=1053.699,78.666,-78.972,171.153,32.458,156.081
C01741=1053.693,78.417,-78.954,171.151,32.456,156.080
C01742=1053.686,78.131,-78.933,171.149,32.454,156.080
C01743=1053.678,77.846,-78.912,171.148,32.451,156.080
C01744=1053.672,77.560,-78.891,171.146,32.449,156.079
C01745=1053.665,77.275,-78.870,171.145,32.446,156.079
C01746=1053.658,77.025,-78.852,171.143,32.444,156.078
C01747=1053.653,76.777,-78.834,171.141,32.442,156.078
C01748=1053.647,76.527,-78.816,171.140,32.439,156.078
C01749=1053.640,76.278,-78.798,171.138,32.437,156.077
C01750=1053.634,76.028,-78.780,171.136,32.435,156.077
C01751=1053.628,75.780,-78.761,171.135,32.433,156.077
C01752=1053.622,75.530,-78.743,171.133,32.431,156.076
C01753=1053.616,75.280,-78.725,171.132,32.428,156.076
C01754=1053.609,75.032,-78.708,171.130,32.426,156.076
C01755=1053.603,74.783,-78.690,171.128,32.424,156.075
C01756=1053.597,74.533,-78.671,171.127,32.421,156.075
C01757=1053.591,74.284,-78.653,171.125,32.419,156.075
C01758=1053.585,74.035,-78.636,171.123,32.417,156.074
C01759=1053.579,73.786,-78.617,171.122,32.415,156.074
C01760=1053.573,73.536,-78.599,171.120,32.413,156.073
C01761=1053.567,73.287,-78.582,171.118,32.410,156.073
C01762=1053.561,73.038,-78.563,171.117,32.408,156.073
C01763=1053.555,72.788,-78.545,171.116,32.406,156.072
C01764=1053.549,72.539,-78.527,171.114,32.404,156.072
C01765=1053.543,72.290,-78.509,171.113,32.402,156.072
C01766=1053.536,72.040,-78.491,171.111,32.399,156.071
C01767=1053.530,71.791,-78.474,171.109,32.397,156.071
C01768=1053.524,71.542,-78.455,171.108,32.395,156.071
C01769=1053.518,71.292,-78.437,171.106,32.392,156.070
C01770=1053.512,71.043,-78.420,171.104,32.390,156.070
C01771=1053.506,70.794,-78.402,171.103,32.388,156.069
C01772=1053.500,70.544,-78.383,171.101,32.386,156.069
C01773=1053.494,70.295,-78.366,171.100,32.384,156.069
C01774=1053.487,70.046,-78.348,171.098,32.381,156.068
C01775=1053.481,69.796,-78.330,171.096,32.379,156.068
C01776=1053.475,69.548,-78.312,171.095,32.377,156.068
C01777=1053.469,69.298,-78.294,171.093,32.375,156.067
C01778=1053.464,69.049,-78.276,171.091,32.373,156.067
C01779=1053.457,68.800,-78.259,171.090,32.370,156.067
C01780=1053.451,68.550,-78.241,171.088,32.368,156.066
C01781=1053.445,68.301,-78.223,171.087,32.366,156.066
C01782=1053.439,68.052,-78.205,171.086,32.363,156.066
C01783=1053.432,67.802,-78.188,171.084,32.361,156.065
C01784=1053.426,67.553,-78.170,171.082,32.359,156.065
C01785=1053.420,67.304,-78.152,171.081,32.357,156.065
C01786=1053.415,67.054,-78.135,171.079,32.355,156.064
C01787=1053.408,66.806,-78.117,171.077,32.353,156.064
C01788=1053.401,66.556,-78.099,171.076,32.350,156.064
C01789=1053.396,66.307,-78.081,171.074,32.348,156.063
C01790=1053.389,66.057,-78.064,171.072,32.346,156.063
C01791=1053.384,65.808,-78.046,171.071,32.343,156.063
C01792=1053.377,65.559,-78.028,171.069,32.341,156.062
C01793=1053.371,65.309,-78.011,171.068,32.340,156.062
C01794=1053.365,65.060,-77.993,171.066,32.337,156.061
C01795=1053.359,64.810,-77.975,171.064,32.335,156.061
C01796=1053.353,64.562,-77.958,171.063,32.333,156.061
